REGION Network 32: Sim Bồn 3: Giới hạn mức nước tối thiểu
   RUNG wire#powerrail
      Contact( "AI_HMI_Sim_Mode" )
      { S7_Templates := "SrcType := Real" } LT_Contact(in1 := "AI_LT3213_Bon3_HMI", in2 := 0.0)
      { S7_GenerateENO := "TRUE" } Move(in := 0.0, out1 => "AI_LT3213_Bon3_HMI")
   END_RUNG
   // the same network as SCL:
   IF "AI_HMI_Sim_Mode" AND ("AI_LT3213_Bon3_HMI" < 0.0) THEN "AI_LT3213_Bon3_HMI" := 0.0; END_IF;
END_REGION

REGION Network 33: Sim Bồn 4: Tăng FQ và LT khi dosing
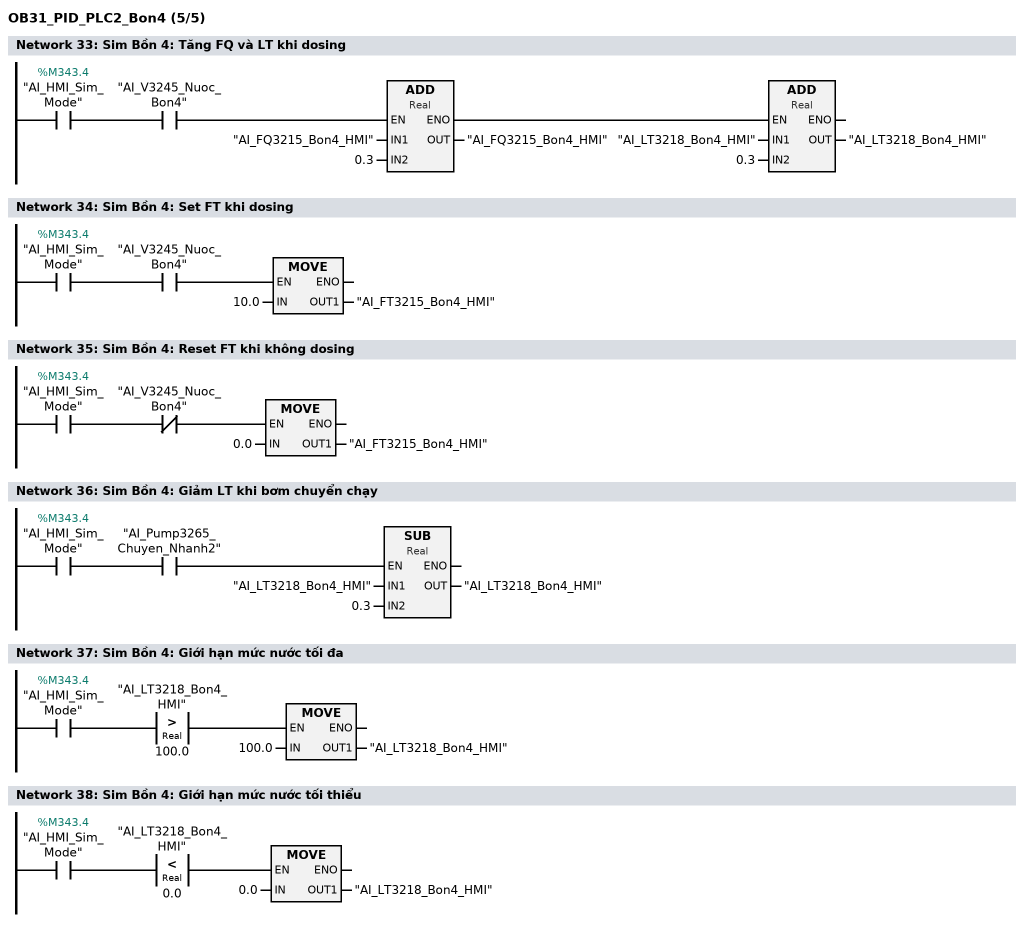
   RUNG wire#powerrail
      Contact( "AI_HMI_Sim_Mode" )
      Contact( "AI_V3245_Nuoc_Bon4" )
      { S7_Templates := "SrcType := Real"; S7_GenerateENO := "TRUE" } Add(in1 := "AI_FQ3215_Bon4_HMI", in2 := 0.3, out => "AI_FQ3215_Bon4_HMI")
      { S7_Templates := "SrcType := Real"; S7_GenerateENO := "TRUE" } Add(in1 := "AI_LT3218_Bon4_HMI", in2 := 0.3, out => "AI_LT3218_Bon4_HMI")
   END_RUNG
   // the same network as SCL:
   // ENO of a box is taken as its EN; it also drops when the box reports an error
   IF "AI_HMI_Sim_Mode" AND "AI_V3245_Nuoc_Bon4" THEN
       "AI_FQ3215_Bon4_HMI" := "AI_FQ3215_Bon4_HMI" + 0.3;
       "AI_LT3218_Bon4_HMI" := "AI_LT3218_Bon4_HMI" + 0.3;
   END_IF;
END_REGION

REGION Network 34: Sim Bồn 4: Set FT khi dosing
   RUNG wire#powerrail
      Contact( "AI_HMI_Sim_Mode" )
      Contact( "AI_V3245_Nuoc_Bon4" )
      { S7_GenerateENO := "TRUE" } Move(in := 10.0, out1 => "AI_FT3215_Bon4_HMI")
   END_RUNG
   // the same network as SCL:
   IF "AI_HMI_Sim_Mode" AND "AI_V3245_Nuoc_Bon4" THEN "AI_FT3215_Bon4_HMI" := 10.0; END_IF;
END_REGION

REGION Network 35: Sim Bồn 4: Reset FT khi không dosing
   RUNG wire#powerrail
      Contact( "AI_HMI_Sim_Mode" )
      I_Contact( "AI_V3245_Nuoc_Bon4" )
      { S7_GenerateENO := "TRUE" } Move(in := 0.0, out1 => "AI_FT3215_Bon4_HMI")
   END_RUNG
   // the same network as SCL:
   IF "AI_HMI_Sim_Mode" AND NOT "AI_V3245_Nuoc_Bon4" THEN "AI_FT3215_Bon4_HMI" := 0.0; END_IF;
END_REGION

REGION Network 36: Sim Bồn 4: Giảm LT khi bơm chuyển chạy
   RUNG wire#powerrail
      Contact( "AI_HMI_Sim_Mode" )
      Contact( "AI_Pump3265_Chuyen_Nhanh2" )
      { S7_Templates := "SrcType := Real"; S7_GenerateENO := "TRUE" } Sub(in1 := "AI_LT3218_Bon4_HMI", in2 := 0.3, out => "AI_LT3218_Bon4_HMI")
   END_RUNG
   // the same network as SCL:
   IF "AI_HMI_Sim_Mode" AND "AI_Pump3265_Chuyen_Nhanh2" THEN
       "AI_LT3218_Bon4_HMI" := "AI_LT3218_Bon4_HMI" - 0.3;
   END_IF;
END_REGION

REGION Network 37: Sim Bồn 4: Giới hạn mức nước tối đa
   RUNG wire#powerrail
      Contact( "AI_HMI_Sim_Mode" )
      { S7_Templates := "SrcType := Real" } GT_Contact(in1 := "AI_LT3218_Bon4_HMI", in2 := 100.0)
      { S7_GenerateENO := "TRUE" } Move(in := 100.0, out1 => "AI_LT3218_Bon4_HMI")
   END_RUNG
   // the same network as SCL:
   IF "AI_HMI_Sim_Mode" AND ("AI_LT3218_Bon4_HMI" > 100.0) THEN "AI_LT3218_Bon4_HMI" := 100.0; END_IF;
END_REGION

REGION Network 38: Sim Bồn 4: Giới hạn mức nước tối thiểu
   RUNG wire#powerrail
      Contact( "AI_HMI_Sim_Mode" )
      { S7_Templates := "SrcType := Real" } LT_Contact(in1 := "AI_LT3218_Bon4_HMI", in2 := 0.0)
      { S7_GenerateENO := "TRUE" } Move(in := 0.0, out1 => "AI_LT3218_Bon4_HMI")
   END_RUNG
   // the same network as SCL:
   IF "AI_HMI_Sim_Mode" AND ("AI_LT3218_Bon4_HMI" < 0.0) THEN "AI_LT3218_Bon4_HMI" := 0.0; END_IF;
END_REGION
END_ORGANIZATION_BLOCK

ORGANIZATION_BLOCK "Cyclic interrupt"   // OB30, LAD, CyclicInterrupt
{ S7_Optimized_Access := 'TRUE' }
VERSION : 0.1
// stored: AutoNumber true, IsIECCheckEnabled false, SetENOAutomatically false
   VAR_INPUT
      Initial_Call : Bool;   // Initial call of this OB
      Event_Count : Int;   // Events discarded
   END_VAR
BEGIN

REGION Network 1
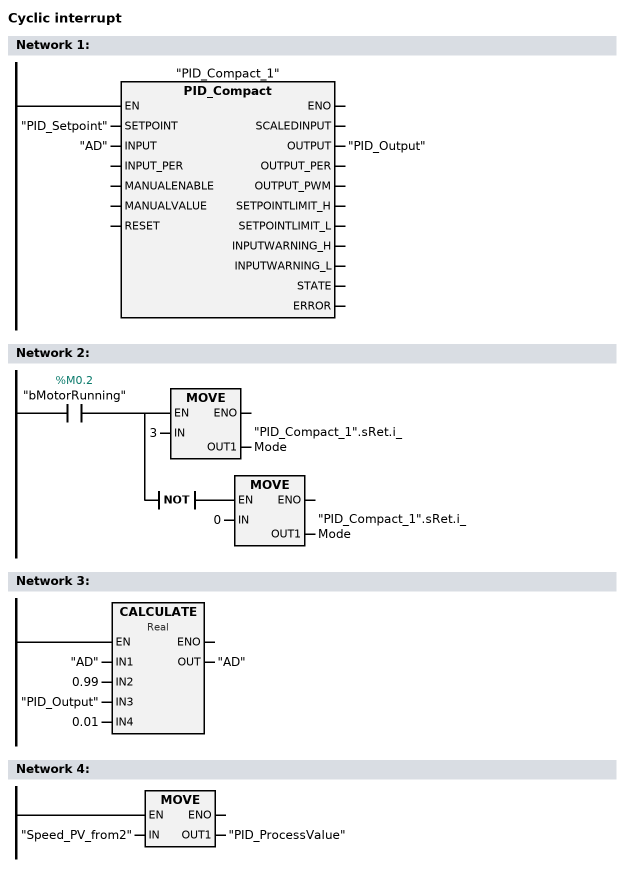
   RUNG wire#powerrail
      "PID_Compact_1".PID_Compact(Setpoint := "PID_Setpoint", Input := "AD", Input_PER :=, ManualEnable :=, ManualValue :=, Reset :=, ScaledInput =>, Output => "PID_Output", Output_PER =>, Output_PWM =>, SetpointLimit_H =>, SetpointLimit_L =>, InputWarning_H =>, InputWarning_L =>, State =>, Error =>)
   END_RUNG
   // the same network as SCL:
   "PID_Compact_1"(Setpoint := "PID_Setpoint", Input := "AD", Output => "PID_Output");   // PID_Compact
END_REGION

REGION Network 2
   RUNG wire#powerrail
      Contact( "bMotorRunning" )
      wire#w1
      Move(in := 3, out1 => "PID_Compact_1".sRet.i_Mode)
   END_RUNG
   RUNG wire#w1
      Not()
      Move(in := 0, out1 => "PID_Compact_1".sRet.i_Mode)
   END_RUNG
   // the same network as SCL:
   IF "bMotorRunning" THEN "PID_Compact_1".sRet.i_Mode := 3; END_IF;
   IF NOT "bMotorRunning" THEN "PID_Compact_1".sRet.i_Mode := 0; END_IF;
END_REGION

REGION Network 3
   RUNG wire#powerrail
      { S7_Templates := "SrcType := Real"; S7_Expression := "IN2*IN1 + IN4*IN3" } Calculate(in1 := "AD", in2 := 0.99, in3 := "PID_Output", in4 := 0.01, out => "AD")
   END_RUNG
   // the same network as SCL:
   "AD" := 0.99*"AD" + 0.01*"PID_Output";
END_REGION

REGION Network 4
   RUNG wire#powerrail
      Move(in := "Speed_PV_from2", out1 => "PID_ProcessValue")
   END_RUNG
   // the same network as SCL:
   "PID_ProcessValue" := "Speed_PV_from2";
END_REGION
END_ORGANIZATION_BLOCK

ORGANIZATION_BLOCK "OB30_Encoder_100ms"   // OB30, LAD, CyclicInterrupt
{ S7_Optimized_Access := 'TRUE' }
VERSION : 0.1
// stored: AutoNumber true, IsIECCheckEnabled false, SetENOAutomatically false
   VAR_INPUT
      Initial_Call : Bool;   // Initial call of this OB
      Event_Count : Int;   // Events discarded
   END_VAR
BEGIN

REGION Network 1: Đọc giá trị HSC và tính Delta Count
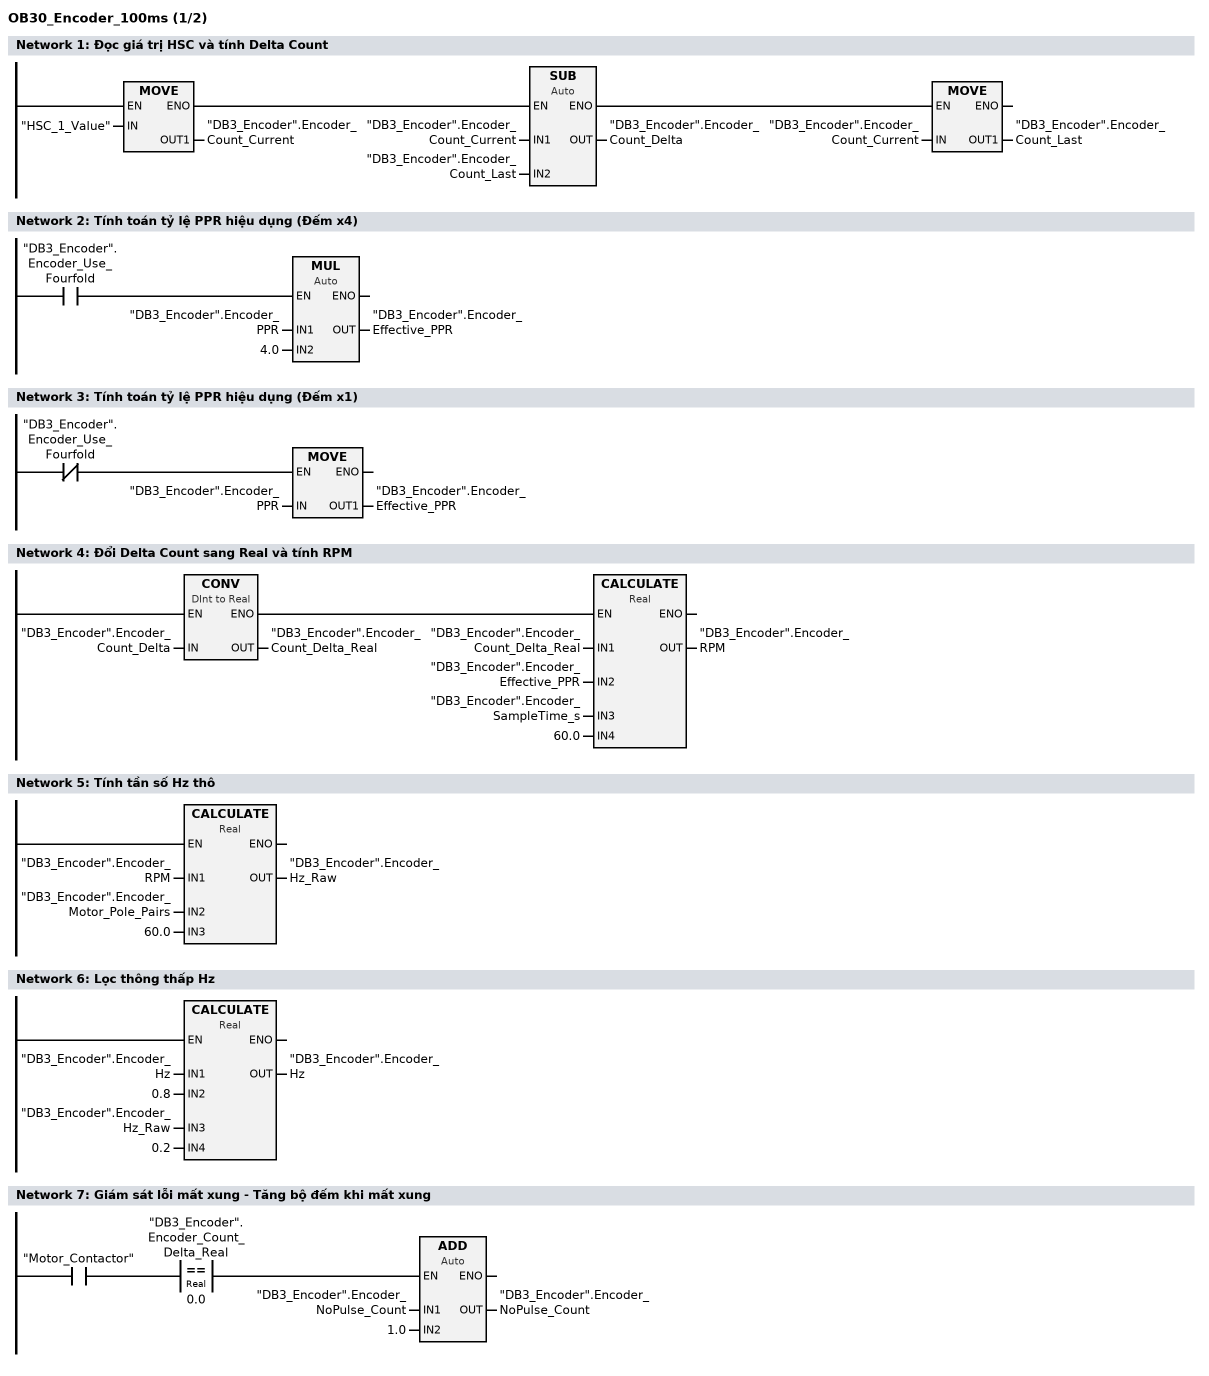
   RUNG wire#powerrail
      { S7_GenerateENO := "TRUE" } Move(in := "HSC_1_Value", out1 => "DB3_Encoder".Encoder_Count_Current)
      { S7_GenerateENO := "TRUE" } Sub(in1 := "DB3_Encoder".Encoder_Count_Current, in2 := "DB3_Encoder".Encoder_Count_Last, out => "DB3_Encoder".Encoder_Count_Delta)
      { S7_GenerateENO := "TRUE" } Move(in := "DB3_Encoder".Encoder_Count_Current, out1 => "DB3_Encoder".Encoder_Count_Last)
   END_RUNG
   // the same network as SCL:
   // ENO of a box is taken as its EN; it also drops when the box reports an error
   "DB3_Encoder".Encoder_Count_Current := "HSC_1_Value";
   "DB3_Encoder".Encoder_Count_Delta := "DB3_Encoder".Encoder_Count_Current - "DB3_Encoder".Encoder_Count_Last;
   "DB3_Encoder".Encoder_Count_Last := "DB3_Encoder".Encoder_Count_Current;
END_REGION

REGION Network 2: Tính toán tỷ lệ PPR hiệu dụng (Đếm x4)
   RUNG wire#powerrail
      Contact( "DB3_Encoder".Encoder_Use_Fourfold )
      { S7_GenerateENO := "TRUE" } Mul(in1 := "DB3_Encoder".Encoder_PPR, in2 := 4.0, out => "DB3_Encoder".Encoder_Effective_PPR)
   END_RUNG
   // the same network as SCL:
   IF "DB3_Encoder".Encoder_Use_Fourfold THEN
       "DB3_Encoder".Encoder_Effective_PPR := "DB3_Encoder".Encoder_PPR * 4.0;
   END_IF;
END_REGION

REGION Network 3: Tính toán tỷ lệ PPR hiệu dụng (Đếm x1)
   RUNG wire#powerrail
      I_Contact( "DB3_Encoder".Encoder_Use_Fourfold )
      { S7_GenerateENO := "TRUE" } Move(in := "DB3_Encoder".Encoder_PPR, out1 => "DB3_Encoder".Encoder_Effective_PPR)
   END_RUNG
   // the same network as SCL:
   IF NOT "DB3_Encoder".Encoder_Use_Fourfold THEN
       "DB3_Encoder".Encoder_Effective_PPR := "DB3_Encoder".Encoder_PPR;
   END_IF;
END_REGION

REGION Network 4: Đổi Delta Count sang Real và tính RPM
   RUNG wire#powerrail
      { S7_Templates := "[SrcType := DInt, DestType := Real]"; S7_GenerateENO := "TRUE" } Convert(in := "DB3_Encoder".Encoder_Count_Delta, out => "DB3_Encoder".Encoder_Count_Delta_Real)
      { S7_Templates := "SrcType := Real"; S7_GenerateENO := "TRUE"; S7_Expression := "(IN1 * IN4) / (IN2 * IN3)" } Calculate(in1 := "DB3_Encoder".Encoder_Count_Delta_Real, in2 := "DB3_Encoder".Encoder_Effective_PPR, in3 := "DB3_Encoder".Encoder_SampleTime_s, in4 := 60.0, out => "DB3_Encoder".Encoder_RPM)
   END_RUNG
   // the same network as SCL:
   // ENO of a box is taken as its EN; it also drops when the box reports an error
   "DB3_Encoder".Encoder_Count_Delta_Real := DINT_TO_REAL("DB3_Encoder".Encoder_Count_Delta);
   "DB3_Encoder".Encoder_RPM := ("DB3_Encoder".Encoder_Count_Delta_Real * 60.0) / ("DB3_Encoder".Encoder_Effective_PPR * "DB3_Encoder".Encoder_SampleTime_s);
END_REGION

REGION Network 5: Tính tần số Hz thô
   RUNG wire#powerrail
      { S7_Templates := "SrcType := Real"; S7_GenerateENO := "TRUE"; S7_Expression := "(IN1 * IN2) / IN3" } Calculate(in1 := "DB3_Encoder".Encoder_RPM, in2 := "DB3_Encoder".Encoder_Motor_Pole_Pairs, in3 := 60.0, out => "DB3_Encoder".Encoder_Hz_Raw)
   END_RUNG
   // the same network as SCL:
   "DB3_Encoder".Encoder_Hz_Raw := ("DB3_Encoder".Encoder_RPM * "DB3_Encoder".Encoder_Motor_Pole_Pairs) / 60.0;
END_REGION

REGION Network 6: Lọc thông thấp Hz
   RUNG wire#powerrail
      { S7_Templates := "SrcType := Real"; S7_GenerateENO := "TRUE"; S7_Expression := "(IN1 * IN2) + (IN3 * IN4)" } Calculate(in1 := "DB3_Encoder".Encoder_Hz, in2 := 0.8, in3 := "DB3_Encoder".Encoder_Hz_Raw, in4 := 0.2, out => "DB3_Encoder".Encoder_Hz)
   END_RUNG
   // the same network as SCL:
   "DB3_Encoder".Encoder_Hz := ("DB3_Encoder".Encoder_Hz * 0.8) + ("DB3_Encoder".Encoder_Hz_Raw * 0.2);
END_REGION

REGION Network 7: Giám sát lỗi mất xung - Tăng bộ đếm khi mất xung
   RUNG wire#powerrail
      Contact( "Motor_Contactor" )
      { S7_Templates := "SrcType := Real" } EQ_Contact(in1 := "DB3_Encoder".Encoder_Count_Delta_Real, in2 := 0.0)
      { S7_GenerateENO := "TRUE" } Add(in1 := "DB3_Encoder".Encoder_NoPulse_Count, in2 := 1.0, out => "DB3_Encoder".Encoder_NoPulse_Count)
   END_RUNG
   // the same network as SCL:
   IF "Motor_Contactor" AND ("DB3_Encoder".Encoder_Count_Delta_Real = 0.0) THEN
       "DB3_Encoder".Encoder_NoPulse_Count := "DB3_Encoder".Encoder_NoPulse_Count + 1.0;
   END_IF;
END_REGION

REGION Network 8: Giám sát lỗi mất xung - Reset bộ đếm khi có xung
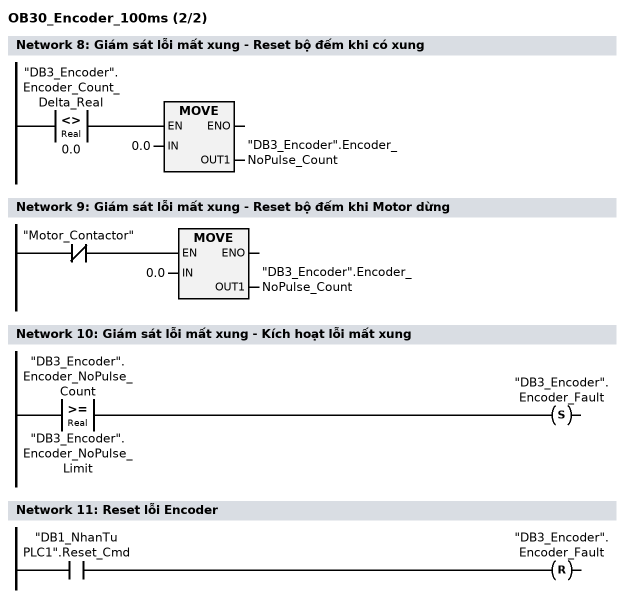
   RUNG wire#powerrail
      { S7_Templates := "SrcType := Real" } NE_Contact(in1 := "DB3_Encoder".Encoder_Count_Delta_Real, in2 := 0.0)
      { S7_GenerateENO := "TRUE" } Move(in := 0.0, out1 => "DB3_Encoder".Encoder_NoPulse_Count)
   END_RUNG
   // the same network as SCL:
   IF "DB3_Encoder".Encoder_Count_Delta_Real <> 0.0 THEN "DB3_Encoder".Encoder_NoPulse_Count := 0.0; END_IF;
END_REGION

REGION Network 9: Giám sát lỗi mất xung - Reset bộ đếm khi Motor dừng
   RUNG wire#powerrail
      I_Contact( "Motor_Contactor" )
      { S7_GenerateENO := "TRUE" } Move(in := 0.0, out1 => "DB3_Encoder".Encoder_NoPulse_Count)
   END_RUNG
   // the same network as SCL:
   IF NOT "Motor_Contactor" THEN "DB3_Encoder".Encoder_NoPulse_Count := 0.0; END_IF;
END_REGION

REGION Network 10: Giám sát lỗi mất xung - Kích hoạt lỗi mất xung
   RUNG wire#powerrail
      { S7_Templates := "SrcType := Real" } GE_Contact(in1 := "DB3_Encoder".Encoder_NoPulse_Count, in2 := "DB3_Encoder".Encoder_NoPulse_Limit)
      S_Coil( "DB3_Encoder".Encoder_Fault )
   END_RUNG
   // the same network as SCL:
   IF "DB3_Encoder".Encoder_NoPulse_Count >= "DB3_Encoder".Encoder_NoPulse_Limit THEN
       "DB3_Encoder".Encoder_Fault := TRUE;
   END_IF;
END_REGION

REGION Network 11: Reset lỗi Encoder
   RUNG wire#powerrail
      Contact( "DB1_NhanTuPLC1".Reset_Cmd )
      R_Coil( "DB3_Encoder".Encoder_Fault )
   END_RUNG
   // the same network as SCL:
   IF "DB1_NhanTuPLC1".Reset_Cmd THEN "DB3_Encoder".Encoder_Fault := FALSE; END_IF;
END_REGION
END_ORGANIZATION_BLOCK

FUNCTION "FC_SCADA_Simulation" : Void   // FC10, LAD
{ S7_Optimized_Access := 'TRUE' }
VERSION : 0.1
// stored: AutoNumber true, IsIECCheckEnabled false
BEGIN

REGION Network 1: Tạo xung kích hoạt chu kỳ mô phỏng (50ms)
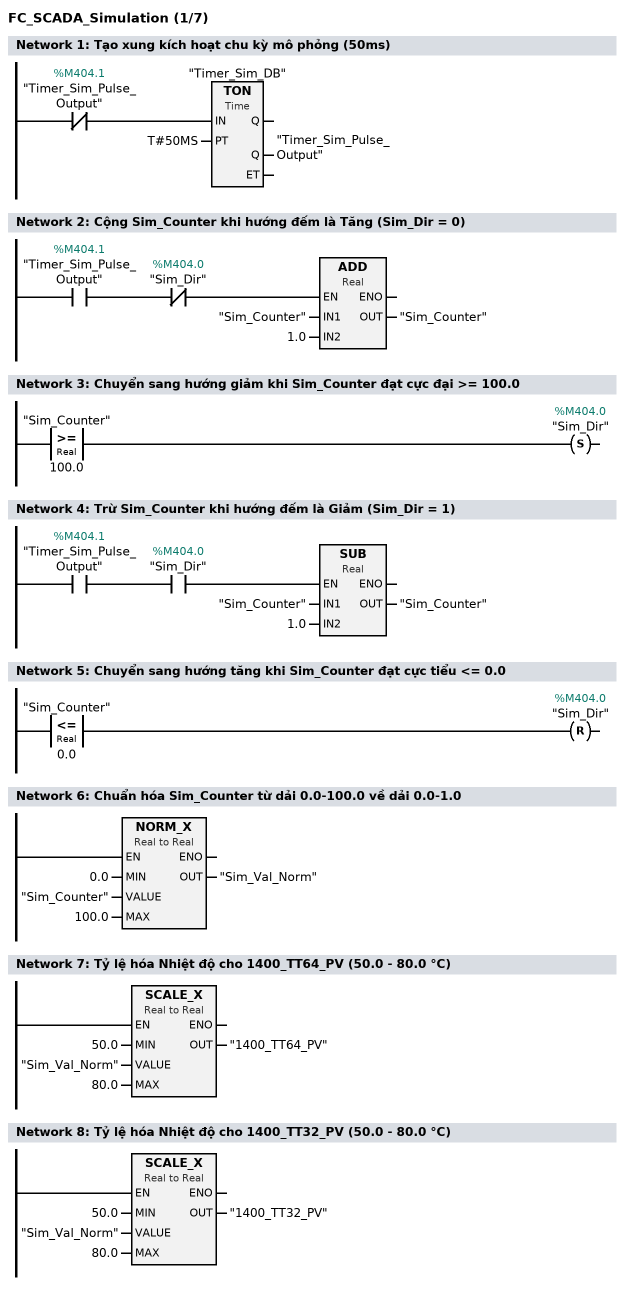
   RUNG wire#powerrail
      I_Contact( "Timer_Sim_Pulse_Output" )
      { S7_Templates := "time_type := Time" } "Timer_Sim_DB".TON(pt := T#50MS, q => "Timer_Sim_Pulse_Output", et =>)
   END_RUNG
   // the same network as SCL:
   "Timer_Sim_DB".TON(IN := NOT "Timer_Sim_Pulse_Output", PT := T#50MS, Q => "Timer_Sim_Pulse_Output");
END_REGION

REGION Network 2: Cộng Sim_Counter khi hướng đếm là Tăng (Sim_Dir = 0)
   RUNG wire#powerrail
      Contact( "Timer_Sim_Pulse_Output" )
      I_Contact( "Sim_Dir" )
      { S7_Templates := "SrcType := Real"; S7_GenerateENO := "TRUE" } Add(in1 := "Sim_Counter", in2 := 1.0, out => "Sim_Counter")
   END_RUNG
   // the same network as SCL:
   IF "Timer_Sim_Pulse_Output" AND NOT "Sim_Dir" THEN "Sim_Counter" := "Sim_Counter" + 1.0; END_IF;
END_REGION

REGION Network 3: Chuyển sang hướng giảm khi Sim_Counter đạt cực đại >= 100.0
   RUNG wire#powerrail
      { S7_Templates := "SrcType := Real" } GE_Contact(in1 := "Sim_Counter", in2 := 100.0)
      S_Coil( "Sim_Dir" )
   END_RUNG
   // the same network as SCL:
   IF "Sim_Counter" >= 100.0 THEN "Sim_Dir" := TRUE; END_IF;
END_REGION

REGION Network 4: Trừ Sim_Counter khi hướng đếm là Giảm (Sim_Dir = 1)
   RUNG wire#powerrail
      Contact( "Timer_Sim_Pulse_Output" )
      Contact( "Sim_Dir" )
      { S7_Templates := "SrcType := Real"; S7_GenerateENO := "TRUE" } Sub(in1 := "Sim_Counter", in2 := 1.0, out => "Sim_Counter")
   END_RUNG
   // the same network as SCL:
   IF "Timer_Sim_Pulse_Output" AND "Sim_Dir" THEN "Sim_Counter" := "Sim_Counter" - 1.0; END_IF;
END_REGION

REGION Network 5: Chuyển sang hướng tăng khi Sim_Counter đạt cực tiểu <= 0.0
   RUNG wire#powerrail
      { S7_Templates := "SrcType := Real" } LE_Contact(in1 := "Sim_Counter", in2 := 0.0)
      R_Coil( "Sim_Dir" )
   END_RUNG
   // the same network as SCL:
   IF "Sim_Counter" <= 0.0 THEN "Sim_Dir" := FALSE; END_IF;
END_REGION

REGION Network 6: Chuẩn hóa Sim_Counter từ dải 0.0-100.0 về dải 0.0-1.0
   RUNG wire#powerrail
      { S7_Templates := "[SrcType := Real, DestType := Real]" } Normalize(min := 0.0, value := "Sim_Counter", max := 100.0, out => "Sim_Val_Norm")
   END_RUNG
   // the same network as SCL:
   "Sim_Val_Norm" := NORM_X(MIN := 0.0, VALUE := "Sim_Counter", MAX := 100.0);
END_REGION

REGION Network 7: Tỷ lệ hóa Nhiệt độ cho 1400_TT64_PV (50.0 - 80.0 °C)
   RUNG wire#powerrail
      { S7_Templates := "[SrcType := Real, DestType := Real]" } Scale(min := 50.0, value := "Sim_Val_Norm", max := 80.0, out => "1400_TT64_PV")
   END_RUNG
   // the same network as SCL:
   "1400_TT64_PV" := SCALE_X(MIN := 50.0, VALUE := "Sim_Val_Norm", MAX := 80.0);
END_REGION

REGION Network 8: Tỷ lệ hóa Nhiệt độ cho 1400_TT32_PV (50.0 - 80.0 °C)
   RUNG wire#powerrail
      { S7_Templates := "[SrcType := Real, DestType := Real]" } Scale(min := 50.0, value := "Sim_Val_Norm", max := 80.0, out => "1400_TT32_PV")
   END_RUNG
   // the same network as SCL:
   "1400_TT32_PV" := SCALE_X(MIN := 50.0, VALUE := "Sim_Val_Norm", MAX := 80.0);
END_REGION

REGION Network 9: Tỷ lệ hóa Nhiệt độ cho 1400_TT101_PV (50.0 - 80.0 °C)
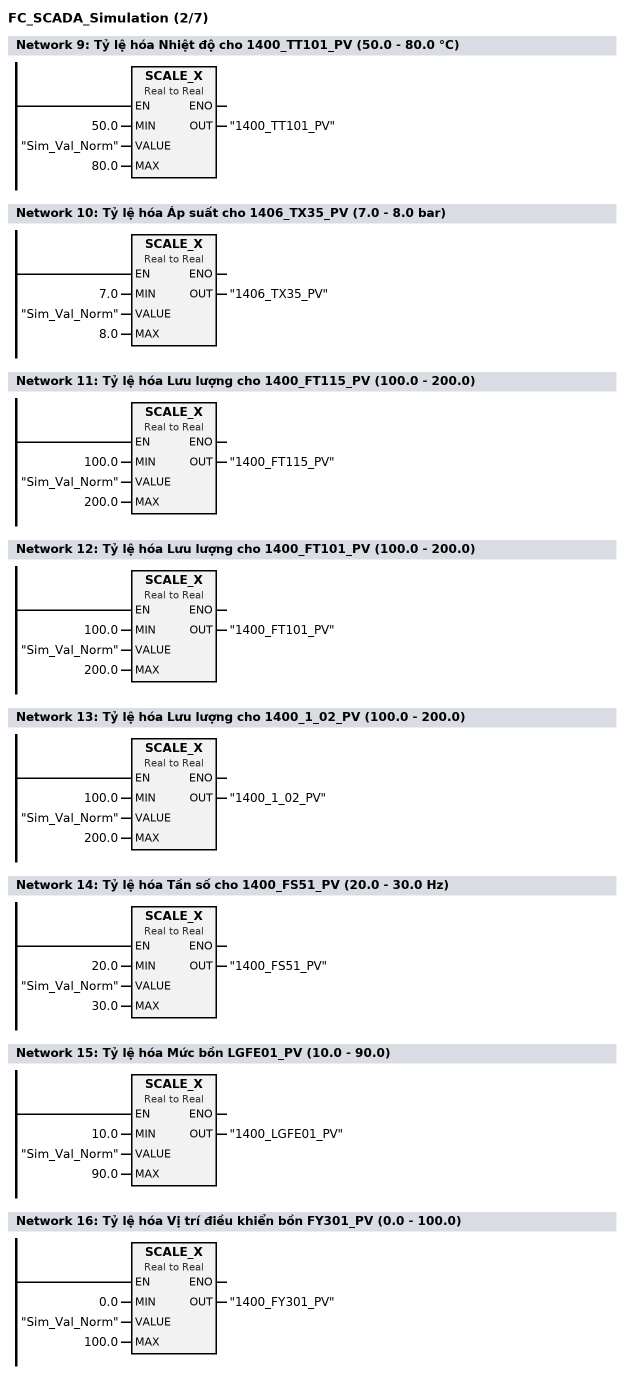
   RUNG wire#powerrail
      { S7_Templates := "[SrcType := Real, DestType := Real]" } Scale(min := 50.0, value := "Sim_Val_Norm", max := 80.0, out => "1400_TT101_PV")
   END_RUNG
   // the same network as SCL:
   "1400_TT101_PV" := SCALE_X(MIN := 50.0, VALUE := "Sim_Val_Norm", MAX := 80.0);
END_REGION

REGION Network 10: Tỷ lệ hóa Áp suất cho 1406_TX35_PV (7.0 - 8.0 bar)
   RUNG wire#powerrail
      { S7_Templates := "[SrcType := Real, DestType := Real]" } Scale(min := 7.0, value := "Sim_Val_Norm", max := 8.0, out => "1406_TX35_PV")
   END_RUNG
   // the same network as SCL:
   "1406_TX35_PV" := SCALE_X(MIN := 7.0, VALUE := "Sim_Val_Norm", MAX := 8.0);
END_REGION

REGION Network 11: Tỷ lệ hóa Lưu lượng cho 1400_FT115_PV (100.0 - 200.0)
   RUNG wire#powerrail
      { S7_Templates := "[SrcType := Real, DestType := Real]" } Scale(min := 100.0, value := "Sim_Val_Norm", max := 200.0, out => "1400_FT115_PV")
   END_RUNG
   // the same network as SCL:
   "1400_FT115_PV" := SCALE_X(MIN := 100.0, VALUE := "Sim_Val_Norm", MAX := 200.0);
END_REGION

REGION Network 12: Tỷ lệ hóa Lưu lượng cho 1400_FT101_PV (100.0 - 200.0)
   RUNG wire#powerrail
      { S7_Templates := "[SrcType := Real, DestType := Real]" } Scale(min := 100.0, value := "Sim_Val_Norm", max := 200.0, out => "1400_FT101_PV")
   END_RUNG
   // the same network as SCL:
   "1400_FT101_PV" := SCALE_X(MIN := 100.0, VALUE := "Sim_Val_Norm", MAX := 200.0);
END_REGION

REGION Network 13: Tỷ lệ hóa Lưu lượng cho 1400_1_02_PV (100.0 - 200.0)
   RUNG wire#powerrail
      { S7_Templates := "[SrcType := Real, DestType := Real]" } Scale(min := 100.0, value := "Sim_Val_Norm", max := 200.0, out => "1400_1_02_PV")
   END_RUNG
   // the same network as SCL:
   "1400_1_02_PV" := SCALE_X(MIN := 100.0, VALUE := "Sim_Val_Norm", MAX := 200.0);
END_REGION

REGION Network 14: Tỷ lệ hóa Tần số cho 1400_FS51_PV (20.0 - 30.0 Hz)
   RUNG wire#powerrail
      { S7_Templates := "[SrcType := Real, DestType := Real]" } Scale(min := 20.0, value := "Sim_Val_Norm", max := 30.0, out => "1400_FS51_PV")
   END_RUNG
   // the same network as SCL:
   "1400_FS51_PV" := SCALE_X(MIN := 20.0, VALUE := "Sim_Val_Norm", MAX := 30.0);
END_REGION

REGION Network 15: Tỷ lệ hóa Mức bồn LGFE01_PV (10.0 - 90.0)
   RUNG wire#powerrail
      { S7_Templates := "[SrcType := Real, DestType := Real]" } Scale(min := 10.0, value := "Sim_Val_Norm", max := 90.0, out => "1400_LGFE01_PV")
   END_RUNG
   // the same network as SCL:
   "1400_LGFE01_PV" := SCALE_X(MIN := 10.0, VALUE := "Sim_Val_Norm", MAX := 90.0);
END_REGION

REGION Network 16: Tỷ lệ hóa Vị trí điều khiển bồn FY301_PV (0.0 - 100.0)
   RUNG wire#powerrail
      { S7_Templates := "[SrcType := Real, DestType := Real]" } Scale(min := 0.0, value := "Sim_Val_Norm", max := 100.0, out => "1400_FY301_PV")
   END_RUNG
   // the same network as SCL:
   "1400_FY301_PV" := SCALE_X(MIN := 0.0, VALUE := "Sim_Val_Norm", MAX := 100.0);
END_REGION

REGION Network 17: Tỷ lệ hóa FTT02_PV (40.0 - 70.0)
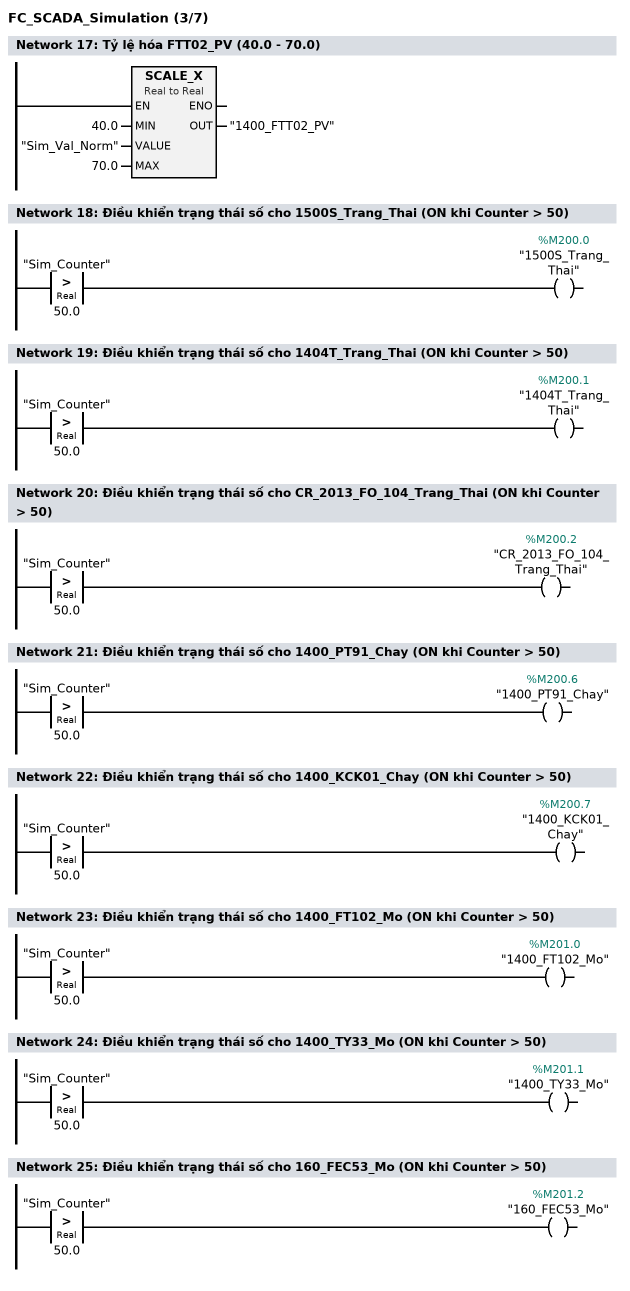
   RUNG wire#powerrail
      { S7_Templates := "[SrcType := Real, DestType := Real]" } Scale(min := 40.0, value := "Sim_Val_Norm", max := 70.0, out => "1400_FTT02_PV")
   END_RUNG
   // the same network as SCL:
   "1400_FTT02_PV" := SCALE_X(MIN := 40.0, VALUE := "Sim_Val_Norm", MAX := 70.0);
END_REGION

REGION Network 18: Điều khiển trạng thái số cho 1500S_Trang_Thai (ON khi Counter > 50)
   RUNG wire#powerrail
      { S7_Templates := "SrcType := Real" } GT_Contact(in1 := "Sim_Counter", in2 := 50.0)
      Coil( "1500S_Trang_Thai" )
   END_RUNG
   // the same network as SCL:
   "1500S_Trang_Thai" := "Sim_Counter" > 50.0;
END_REGION

REGION Network 19: Điều khiển trạng thái số cho 1404T_Trang_Thai (ON khi Counter > 50)
   RUNG wire#powerrail
      { S7_Templates := "SrcType := Real" } GT_Contact(in1 := "Sim_Counter", in2 := 50.0)
      Coil( "1404T_Trang_Thai" )
   END_RUNG
   // the same network as SCL:
   "1404T_Trang_Thai" := "Sim_Counter" > 50.0;
END_REGION

REGION Network 20: Điều khiển trạng thái số cho CR_2013_FO_104_Trang_Thai (ON khi Counter > 50)
   RUNG wire#powerrail
      { S7_Templates := "SrcType := Real" } GT_Contact(in1 := "Sim_Counter", in2 := 50.0)
      Coil( "CR_2013_FO_104_Trang_Thai" )
   END_RUNG
   // the same network as SCL:
   "CR_2013_FO_104_Trang_Thai" := "Sim_Counter" > 50.0;
END_REGION

REGION Network 21: Điều khiển trạng thái số cho 1400_PT91_Chay (ON khi Counter > 50)
   RUNG wire#powerrail
      { S7_Templates := "SrcType := Real" } GT_Contact(in1 := "Sim_Counter", in2 := 50.0)
      Coil( "1400_PT91_Chay" )
   END_RUNG
   // the same network as SCL:
   "1400_PT91_Chay" := "Sim_Counter" > 50.0;
END_REGION

REGION Network 22: Điều khiển trạng thái số cho 1400_KCK01_Chay (ON khi Counter > 50)
   RUNG wire#powerrail
      { S7_Templates := "SrcType := Real" } GT_Contact(in1 := "Sim_Counter", in2 := 50.0)
      Coil( "1400_KCK01_Chay" )
   END_RUNG
   // the same network as SCL:
   "1400_KCK01_Chay" := "Sim_Counter" > 50.0;
END_REGION

REGION Network 23: Điều khiển trạng thái số cho 1400_FT102_Mo (ON khi Counter > 50)
   RUNG wire#powerrail
      { S7_Templates := "SrcType := Real" } GT_Contact(in1 := "Sim_Counter", in2 := 50.0)
      Coil( "1400_FT102_Mo" )
   END_RUNG
   // the same network as SCL:
   "1400_FT102_Mo" := "Sim_Counter" > 50.0;
END_REGION

REGION Network 24: Điều khiển trạng thái số cho 1400_TY33_Mo (ON khi Counter > 50)
   RUNG wire#powerrail
      { S7_Templates := "SrcType := Real" } GT_Contact(in1 := "Sim_Counter", in2 := 50.0)
      Coil( "1400_TY33_Mo" )
   END_RUNG
   // the same network as SCL:
   "1400_TY33_Mo" := "Sim_Counter" > 50.0;
END_REGION

REGION Network 25: Điều khiển trạng thái số cho 160_FEC53_Mo (ON khi Counter > 50)
   RUNG wire#powerrail
      { S7_Templates := "SrcType := Real" } GT_Contact(in1 := "Sim_Counter", in2 := 50.0)
      Coil( "160_FEC53_Mo" )
   END_RUNG
   // the same network as SCL:
   "160_FEC53_Mo" := "Sim_Counter" > 50.0;
END_REGION

REGION Network 26: Điều khiển trạng thái số cho BFOC_SS_20_06_Trang_Thai (ON khi Counter <= 50)
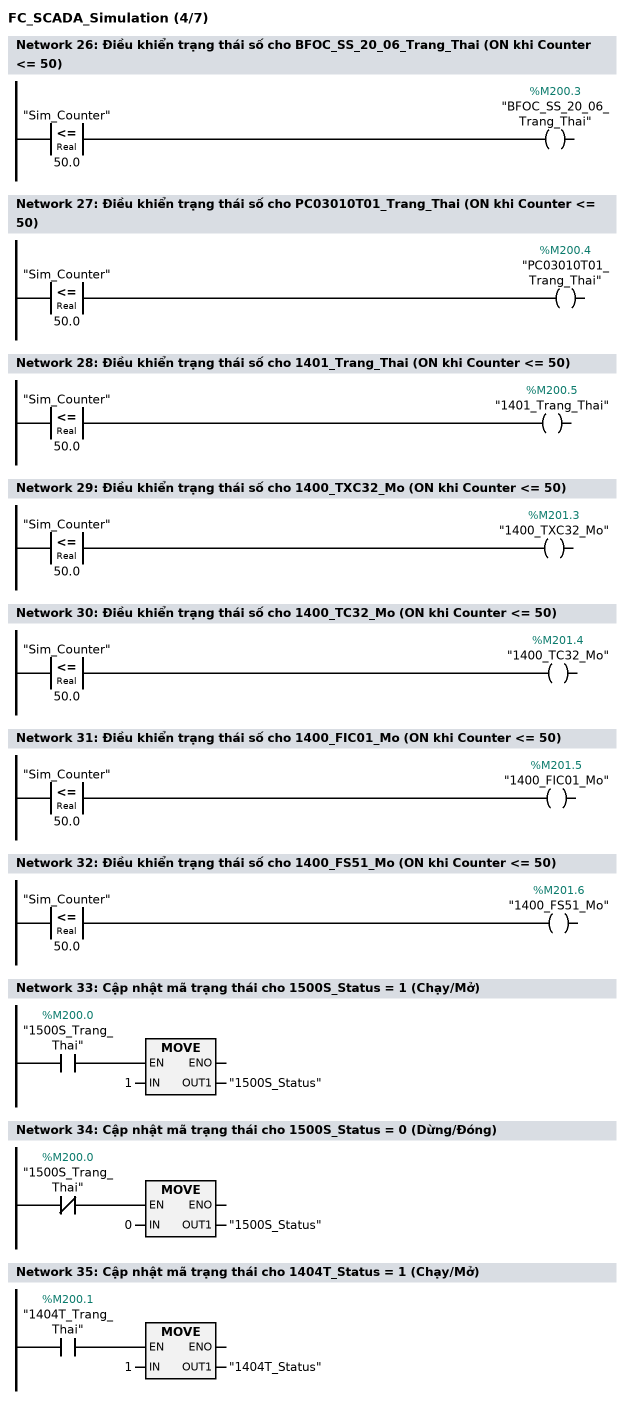
   RUNG wire#powerrail
      { S7_Templates := "SrcType := Real" } LE_Contact(in1 := "Sim_Counter", in2 := 50.0)
      Coil( "BFOC_SS_20_06_Trang_Thai" )
   END_RUNG
   // the same network as SCL:
   "BFOC_SS_20_06_Trang_Thai" := "Sim_Counter" <= 50.0;
END_REGION

REGION Network 27: Điều khiển trạng thái số cho PC03010T01_Trang_Thai (ON khi Counter <= 50)
   RUNG wire#powerrail
      { S7_Templates := "SrcType := Real" } LE_Contact(in1 := "Sim_Counter", in2 := 50.0)
      Coil( "PC03010T01_Trang_Thai" )
   END_RUNG
   // the same network as SCL:
   "PC03010T01_Trang_Thai" := "Sim_Counter" <= 50.0;
END_REGION

REGION Network 28: Điều khiển trạng thái số cho 1401_Trang_Thai (ON khi Counter <= 50)
   RUNG wire#powerrail
      { S7_Templates := "SrcType := Real" } LE_Contact(in1 := "Sim_Counter", in2 := 50.0)
      Coil( "1401_Trang_Thai" )
   END_RUNG
   // the same network as SCL:
   "1401_Trang_Thai" := "Sim_Counter" <= 50.0;
END_REGION

REGION Network 29: Điều khiển trạng thái số cho 1400_TXC32_Mo (ON khi Counter <= 50)
   RUNG wire#powerrail
      { S7_Templates := "SrcType := Real" } LE_Contact(in1 := "Sim_Counter", in2 := 50.0)
      Coil( "1400_TXC32_Mo" )
   END_RUNG
   // the same network as SCL:
   "1400_TXC32_Mo" := "Sim_Counter" <= 50.0;
END_REGION

REGION Network 30: Điều khiển trạng thái số cho 1400_TC32_Mo (ON khi Counter <= 50)
   RUNG wire#powerrail
      { S7_Templates := "SrcType := Real" } LE_Contact(in1 := "Sim_Counter", in2 := 50.0)
      Coil( "1400_TC32_Mo" )
   END_RUNG
   // the same network as SCL:
   "1400_TC32_Mo" := "Sim_Counter" <= 50.0;
END_REGION

REGION Network 31: Điều khiển trạng thái số cho 1400_FIC01_Mo (ON khi Counter <= 50)
   RUNG wire#powerrail
      { S7_Templates := "SrcType := Real" } LE_Contact(in1 := "Sim_Counter", in2 := 50.0)
      Coil( "1400_FIC01_Mo" )
   END_RUNG
   // the same network as SCL:
   "1400_FIC01_Mo" := "Sim_Counter" <= 50.0;
END_REGION

REGION Network 32: Điều khiển trạng thái số cho 1400_FS51_Mo (ON khi Counter <= 50)
   RUNG wire#powerrail
      { S7_Templates := "SrcType := Real" } LE_Contact(in1 := "Sim_Counter", in2 := 50.0)
      Coil( "1400_FS51_Mo" )
   END_RUNG
   // the same network as SCL:
   "1400_FS51_Mo" := "Sim_Counter" <= 50.0;
END_REGION

REGION Network 33: Cập nhật mã trạng thái cho 1500S_Status = 1 (Chạy/Mở)
   RUNG wire#powerrail
      Contact( "1500S_Trang_Thai" )
      { S7_GenerateENO := "TRUE" } Move(in := 1, out1 => "1500S_Status")
   END_RUNG
   // the same network as SCL:
   IF "1500S_Trang_Thai" THEN "1500S_Status" := 1; END_IF;
END_REGION

REGION Network 34: Cập nhật mã trạng thái cho 1500S_Status = 0 (Dừng/Đóng)
   RUNG wire#powerrail
      I_Contact( "1500S_Trang_Thai" )
      { S7_GenerateENO := "TRUE" } Move(in := 0, out1 => "1500S_Status")
   END_RUNG
   // the same network as SCL:
   IF NOT "1500S_Trang_Thai" THEN "1500S_Status" := 0; END_IF;
END_REGION

REGION Network 35: Cập nhật mã trạng thái cho 1404T_Status = 1 (Chạy/Mở)
   RUNG wire#powerrail
      Contact( "1404T_Trang_Thai" )
      { S7_GenerateENO := "TRUE" } Move(in := 1, out1 => "1404T_Status")
   END_RUNG
   // the same network as SCL:
   IF "1404T_Trang_Thai" THEN "1404T_Status" := 1; END_IF;
END_REGION

REGION Network 36: Cập nhật mã trạng thái cho 1404T_Status = 0 (Dừng/Đóng)
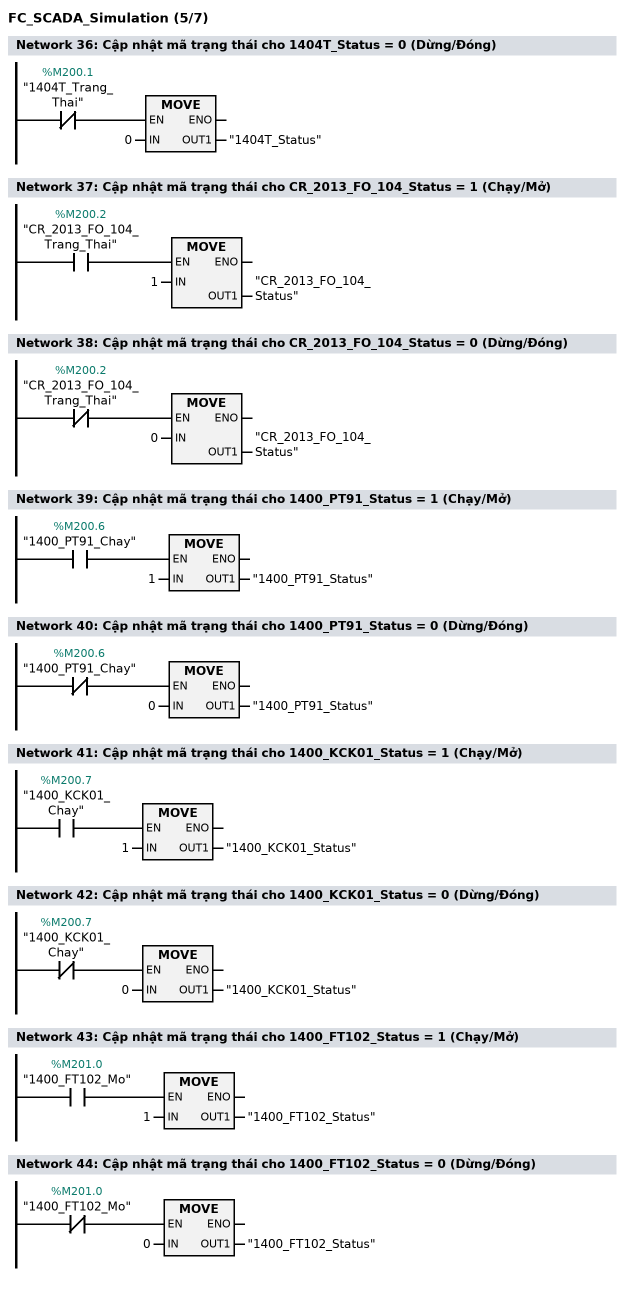
   RUNG wire#powerrail
      I_Contact( "1404T_Trang_Thai" )
      { S7_GenerateENO := "TRUE" } Move(in := 0, out1 => "1404T_Status")
   END_RUNG
   // the same network as SCL:
   IF NOT "1404T_Trang_Thai" THEN "1404T_Status" := 0; END_IF;
END_REGION

REGION Network 37: Cập nhật mã trạng thái cho CR_2013_FO_104_Status = 1 (Chạy/Mở)
   RUNG wire#powerrail
      Contact( "CR_2013_FO_104_Trang_Thai" )
      { S7_GenerateENO := "TRUE" } Move(in := 1, out1 => "CR_2013_FO_104_Status")
   END_RUNG
   // the same network as SCL:
   IF "CR_2013_FO_104_Trang_Thai" THEN "CR_2013_FO_104_Status" := 1; END_IF;
END_REGION

REGION Network 38: Cập nhật mã trạng thái cho CR_2013_FO_104_Status = 0 (Dừng/Đóng)
   RUNG wire#powerrail
      I_Contact( "CR_2013_FO_104_Trang_Thai" )
      { S7_GenerateENO := "TRUE" } Move(in := 0, out1 => "CR_2013_FO_104_Status")
   END_RUNG
   // the same network as SCL:
   IF NOT "CR_2013_FO_104_Trang_Thai" THEN "CR_2013_FO_104_Status" := 0; END_IF;
END_REGION

REGION Network 39: Cập nhật mã trạng thái cho 1400_PT91_Status = 1 (Chạy/Mở)
   RUNG wire#powerrail
      Contact( "1400_PT91_Chay" )
      { S7_GenerateENO := "TRUE" } Move(in := 1, out1 => "1400_PT91_Status")
   END_RUNG
   // the same network as SCL:
   IF "1400_PT91_Chay" THEN "1400_PT91_Status" := 1; END_IF;
END_REGION

REGION Network 40: Cập nhật mã trạng thái cho 1400_PT91_Status = 0 (Dừng/Đóng)
   RUNG wire#powerrail
      I_Contact( "1400_PT91_Chay" )
      { S7_GenerateENO := "TRUE" } Move(in := 0, out1 => "1400_PT91_Status")
   END_RUNG
   // the same network as SCL:
   IF NOT "1400_PT91_Chay" THEN "1400_PT91_Status" := 0; END_IF;
END_REGION

REGION Network 41: Cập nhật mã trạng thái cho 1400_KCK01_Status = 1 (Chạy/Mở)
   RUNG wire#powerrail
      Contact( "1400_KCK01_Chay" )
      { S7_GenerateENO := "TRUE" } Move(in := 1, out1 => "1400_KCK01_Status")
   END_RUNG
   // the same network as SCL:
   IF "1400_KCK01_Chay" THEN "1400_KCK01_Status" := 1; END_IF;
END_REGION

REGION Network 42: Cập nhật mã trạng thái cho 1400_KCK01_Status = 0 (Dừng/Đóng)
   RUNG wire#powerrail
      I_Contact( "1400_KCK01_Chay" )
      { S7_GenerateENO := "TRUE" } Move(in := 0, out1 => "1400_KCK01_Status")
   END_RUNG
   // the same network as SCL:
   IF NOT "1400_KCK01_Chay" THEN "1400_KCK01_Status" := 0; END_IF;
END_REGION

REGION Network 43: Cập nhật mã trạng thái cho 1400_FT102_Status = 1 (Chạy/Mở)
   RUNG wire#powerrail
      Contact( "1400_FT102_Mo" )
      { S7_GenerateENO := "TRUE" } Move(in := 1, out1 => "1400_FT102_Status")
   END_RUNG
   // the same network as SCL:
   IF "1400_FT102_Mo" THEN "1400_FT102_Status" := 1; END_IF;
END_REGION

REGION Network 44: Cập nhật mã trạng thái cho 1400_FT102_Status = 0 (Dừng/Đóng)
   RUNG wire#powerrail
      I_Contact( "1400_FT102_Mo" )
      { S7_GenerateENO := "TRUE" } Move(in := 0, out1 => "1400_FT102_Status")
   END_RUNG
   // the same network as SCL:
   IF NOT "1400_FT102_Mo" THEN "1400_FT102_Status" := 0; END_IF;
END_REGION

REGION Network 45: Cập nhật mã trạng thái cho 1400_TY33_Status = 1 (Chạy/Mở)
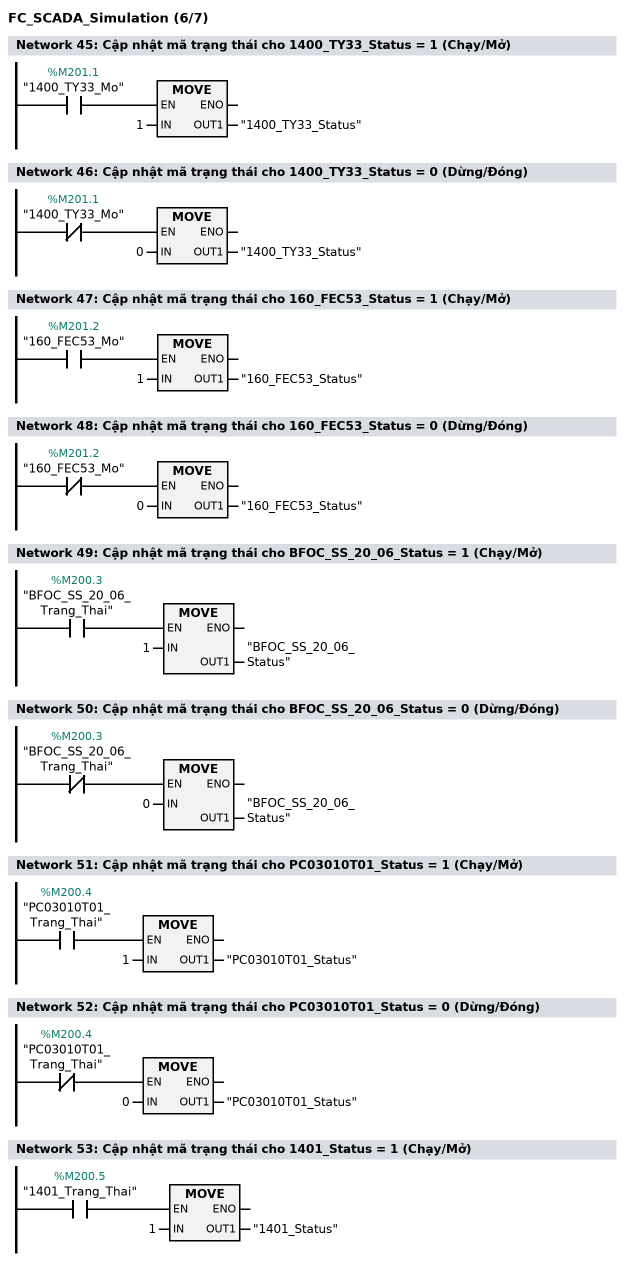
   RUNG wire#powerrail
      Contact( "1400_TY33_Mo" )
      { S7_GenerateENO := "TRUE" } Move(in := 1, out1 => "1400_TY33_Status")
   END_RUNG
   // the same network as SCL:
   IF "1400_TY33_Mo" THEN "1400_TY33_Status" := 1; END_IF;
END_REGION

REGION Network 46: Cập nhật mã trạng thái cho 1400_TY33_Status = 0 (Dừng/Đóng)
   RUNG wire#powerrail
      I_Contact( "1400_TY33_Mo" )
      { S7_GenerateENO := "TRUE" } Move(in := 0, out1 => "1400_TY33_Status")
   END_RUNG
   // the same network as SCL:
   IF NOT "1400_TY33_Mo" THEN "1400_TY33_Status" := 0; END_IF;
END_REGION

REGION Network 47: Cập nhật mã trạng thái cho 160_FEC53_Status = 1 (Chạy/Mở)
   RUNG wire#powerrail
      Contact( "160_FEC53_Mo" )
      { S7_GenerateENO := "TRUE" } Move(in := 1, out1 => "160_FEC53_Status")
   END_RUNG
   // the same network as SCL:
   IF "160_FEC53_Mo" THEN "160_FEC53_Status" := 1; END_IF;
END_REGION

REGION Network 48: Cập nhật mã trạng thái cho 160_FEC53_Status = 0 (Dừng/Đóng)
   RUNG wire#powerrail
      I_Contact( "160_FEC53_Mo" )
      { S7_GenerateENO := "TRUE" } Move(in := 0, out1 => "160_FEC53_Status")
   END_RUNG
   // the same network as SCL:
   IF NOT "160_FEC53_Mo" THEN "160_FEC53_Status" := 0; END_IF;
END_REGION

REGION Network 49: Cập nhật mã trạng thái cho BFOC_SS_20_06_Status = 1 (Chạy/Mở)
   RUNG wire#powerrail
      Contact( "BFOC_SS_20_06_Trang_Thai" )
      { S7_GenerateENO := "TRUE" } Move(in := 1, out1 => "BFOC_SS_20_06_Status")
   END_RUNG
   // the same network as SCL:
   IF "BFOC_SS_20_06_Trang_Thai" THEN "BFOC_SS_20_06_Status" := 1; END_IF;
END_REGION

REGION Network 50: Cập nhật mã trạng thái cho BFOC_SS_20_06_Status = 0 (Dừng/Đóng)
   RUNG wire#powerrail
      I_Contact( "BFOC_SS_20_06_Trang_Thai" )
      { S7_GenerateENO := "TRUE" } Move(in := 0, out1 => "BFOC_SS_20_06_Status")
   END_RUNG
   // the same network as SCL:
   IF NOT "BFOC_SS_20_06_Trang_Thai" THEN "BFOC_SS_20_06_Status" := 0; END_IF;
END_REGION

REGION Network 51: Cập nhật mã trạng thái cho PC03010T01_Status = 1 (Chạy/Mở)
   RUNG wire#powerrail
      Contact( "PC03010T01_Trang_Thai" )
      { S7_GenerateENO := "TRUE" } Move(in := 1, out1 => "PC03010T01_Status")
   END_RUNG
   // the same network as SCL:
   IF "PC03010T01_Trang_Thai" THEN "PC03010T01_Status" := 1; END_IF;
END_REGION

REGION Network 52: Cập nhật mã trạng thái cho PC03010T01_Status = 0 (Dừng/Đóng)
   RUNG wire#powerrail
      I_Contact( "PC03010T01_Trang_Thai" )
      { S7_GenerateENO := "TRUE" } Move(in := 0, out1 => "PC03010T01_Status")
   END_RUNG
   // the same network as SCL:
   IF NOT "PC03010T01_Trang_Thai" THEN "PC03010T01_Status" := 0; END_IF;
END_REGION

REGION Network 53: Cập nhật mã trạng thái cho 1401_Status = 1 (Chạy/Mở)
   RUNG wire#powerrail
      Contact( "1401_Trang_Thai" )
      { S7_GenerateENO := "TRUE" } Move(in := 1, out1 => "1401_Status")
   END_RUNG
   // the same network as SCL:
   IF "1401_Trang_Thai" THEN "1401_Status" := 1; END_IF;
END_REGION

REGION Network 54: Cập nhật mã trạng thái cho 1401_Status = 0 (Dừng/Đóng)
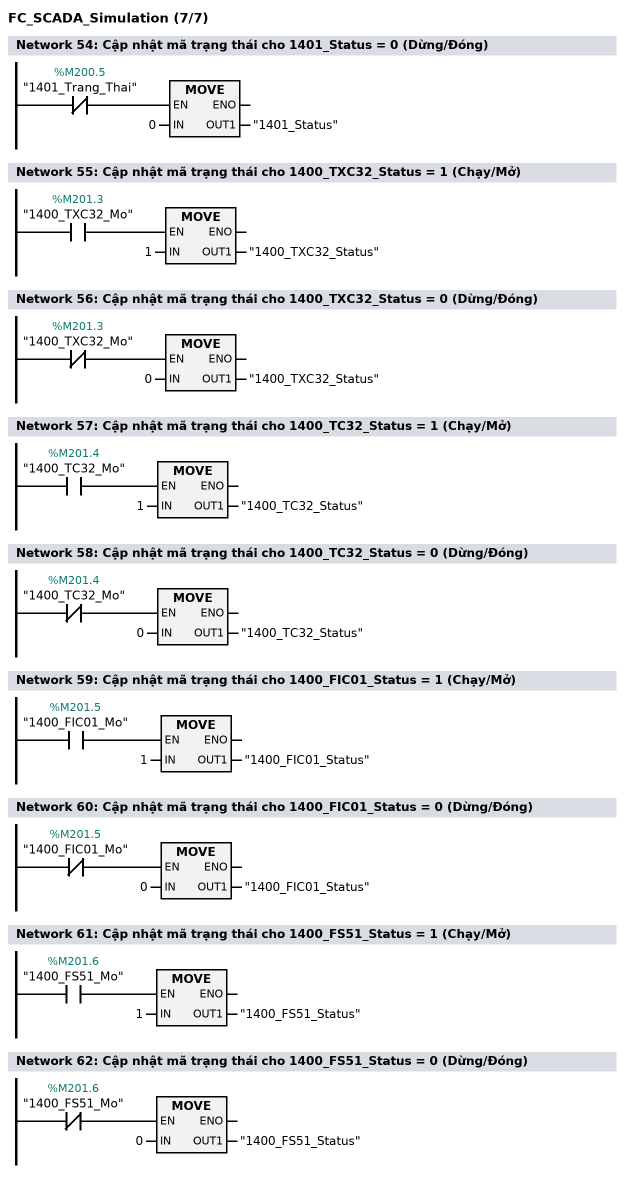
   RUNG wire#powerrail
      I_Contact( "1401_Trang_Thai" )
      { S7_GenerateENO := "TRUE" } Move(in := 0, out1 => "1401_Status")
   END_RUNG
   // the same network as SCL:
   IF NOT "1401_Trang_Thai" THEN "1401_Status" := 0; END_IF;
END_REGION

REGION Network 55: Cập nhật mã trạng thái cho 1400_TXC32_Status = 1 (Chạy/Mở)
   RUNG wire#powerrail
      Contact( "1400_TXC32_Mo" )
      { S7_GenerateENO := "TRUE" } Move(in := 1, out1 => "1400_TXC32_Status")
   END_RUNG
   // the same network as SCL:
   IF "1400_TXC32_Mo" THEN "1400_TXC32_Status" := 1; END_IF;
END_REGION

REGION Network 56: Cập nhật mã trạng thái cho 1400_TXC32_Status = 0 (Dừng/Đóng)
   RUNG wire#powerrail
      I_Contact( "1400_TXC32_Mo" )
      { S7_GenerateENO := "TRUE" } Move(in := 0, out1 => "1400_TXC32_Status")
   END_RUNG
   // the same network as SCL:
   IF NOT "1400_TXC32_Mo" THEN "1400_TXC32_Status" := 0; END_IF;
END_REGION

REGION Network 57: Cập nhật mã trạng thái cho 1400_TC32_Status = 1 (Chạy/Mở)
   RUNG wire#powerrail
      Contact( "1400_TC32_Mo" )
      { S7_GenerateENO := "TRUE" } Move(in := 1, out1 => "1400_TC32_Status")
   END_RUNG
   // the same network as SCL:
   IF "1400_TC32_Mo" THEN "1400_TC32_Status" := 1; END_IF;
END_REGION

REGION Network 58: Cập nhật mã trạng thái cho 1400_TC32_Status = 0 (Dừng/Đóng)
   RUNG wire#powerrail
      I_Contact( "1400_TC32_Mo" )
      { S7_GenerateENO := "TRUE" } Move(in := 0, out1 => "1400_TC32_Status")
   END_RUNG
   // the same network as SCL:
   IF NOT "1400_TC32_Mo" THEN "1400_TC32_Status" := 0; END_IF;
END_REGION

REGION Network 59: Cập nhật mã trạng thái cho 1400_FIC01_Status = 1 (Chạy/Mở)
   RUNG wire#powerrail
      Contact( "1400_FIC01_Mo" )
      { S7_GenerateENO := "TRUE" } Move(in := 1, out1 => "1400_FIC01_Status")
   END_RUNG
   // the same network as SCL:
   IF "1400_FIC01_Mo" THEN "1400_FIC01_Status" := 1; END_IF;
END_REGION

REGION Network 60: Cập nhật mã trạng thái cho 1400_FIC01_Status = 0 (Dừng/Đóng)
   RUNG wire#powerrail
      I_Contact( "1400_FIC01_Mo" )
      { S7_GenerateENO := "TRUE" } Move(in := 0, out1 => "1400_FIC01_Status")
   END_RUNG
   // the same network as SCL:
   IF NOT "1400_FIC01_Mo" THEN "1400_FIC01_Status" := 0; END_IF;
END_REGION

REGION Network 61: Cập nhật mã trạng thái cho 1400_FS51_Status = 1 (Chạy/Mở)
   RUNG wire#powerrail
      Contact( "1400_FS51_Mo" )
      { S7_GenerateENO := "TRUE" } Move(in := 1, out1 => "1400_FS51_Status")
   END_RUNG
   // the same network as SCL:
   IF "1400_FS51_Mo" THEN "1400_FS51_Status" := 1; END_IF;
END_REGION

REGION Network 62: Cập nhật mã trạng thái cho 1400_FS51_Status = 0 (Dừng/Đóng)
   RUNG wire#powerrail
      I_Contact( "1400_FS51_Mo" )
      { S7_GenerateENO := "TRUE" } Move(in := 0, out1 => "1400_FS51_Status")
   END_RUNG
   // the same network as SCL:
   IF NOT "1400_FS51_Mo" THEN "1400_FS51_Status" := 0; END_IF;
END_REGION
END_FUNCTION

BLOCK "WT_Temp_Schema"   // PlcWatchTable
BEGIN
END_BLOCK

BLOCK "WT_Test_Import_DB_Schema"   // PlcWatchTable
BEGIN
END_BLOCK

BLOCK "WT_Test_Import_Schema"   // PlcWatchTable
BEGIN
END_BLOCK

FUNCTION_BLOCK "A_COUNTER"   // FB12, LAD
VERSION : 0.1
// stored: AutoNumber true, IsIECCheckEnabled false, UDAEnableTagReadback false
BEGIN

REGION Network 1
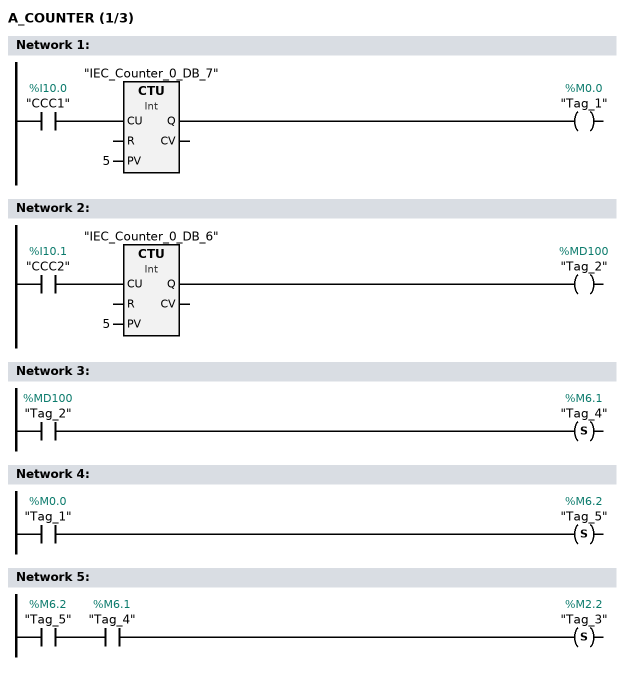
   RUNG wire#powerrail
      Contact( "CCC1" )
      { S7_Templates := "value_type := Int" } "IEC_Counter_0_DB_7".CTU(r :=, pv := 5, cv =>)
      Coil( "Tag_1" )
   END_RUNG
   // the same network as SCL:
   "IEC_Counter_0_DB_7".CTU(CU := "CCC1", PV := 5);
   "Tag_1" := "IEC_Counter_0_DB_7".Q;
END_REGION

REGION Network 2
   RUNG wire#powerrail
      Contact( "CCC2" )
      { S7_Templates := "value_type := Int" } "IEC_Counter_0_DB_6".CTU(r :=, pv := 5, cv =>)
      Coil( "Tag_2" )
   END_RUNG
   // the same network as SCL:
   "IEC_Counter_0_DB_6".CTU(CU := "CCC2", PV := 5);
   "Tag_2" := "IEC_Counter_0_DB_6".Q;
END_REGION

REGION Network 3
   RUNG wire#powerrail
      Contact( "Tag_2" )
      S_Coil( "Tag_4" )
   END_RUNG
   // the same network as SCL:
   IF "Tag_2" THEN "Tag_4" := TRUE; END_IF;
END_REGION

REGION Network 4
   RUNG wire#powerrail
      Contact( "Tag_1" )
      S_Coil( "Tag_5" )
   END_RUNG
   // the same network as SCL:
   IF "Tag_1" THEN "Tag_5" := TRUE; END_IF;
END_REGION

REGION Network 5
   RUNG wire#powerrail
      Contact( "Tag_5" )
      Contact( "Tag_4" )
      S_Coil( "Tag_3" )
   END_RUNG
   // the same network as SCL:
   IF "Tag_5" AND "Tag_4" THEN "Tag_3" := TRUE; END_IF;
END_REGION

REGION Network 6
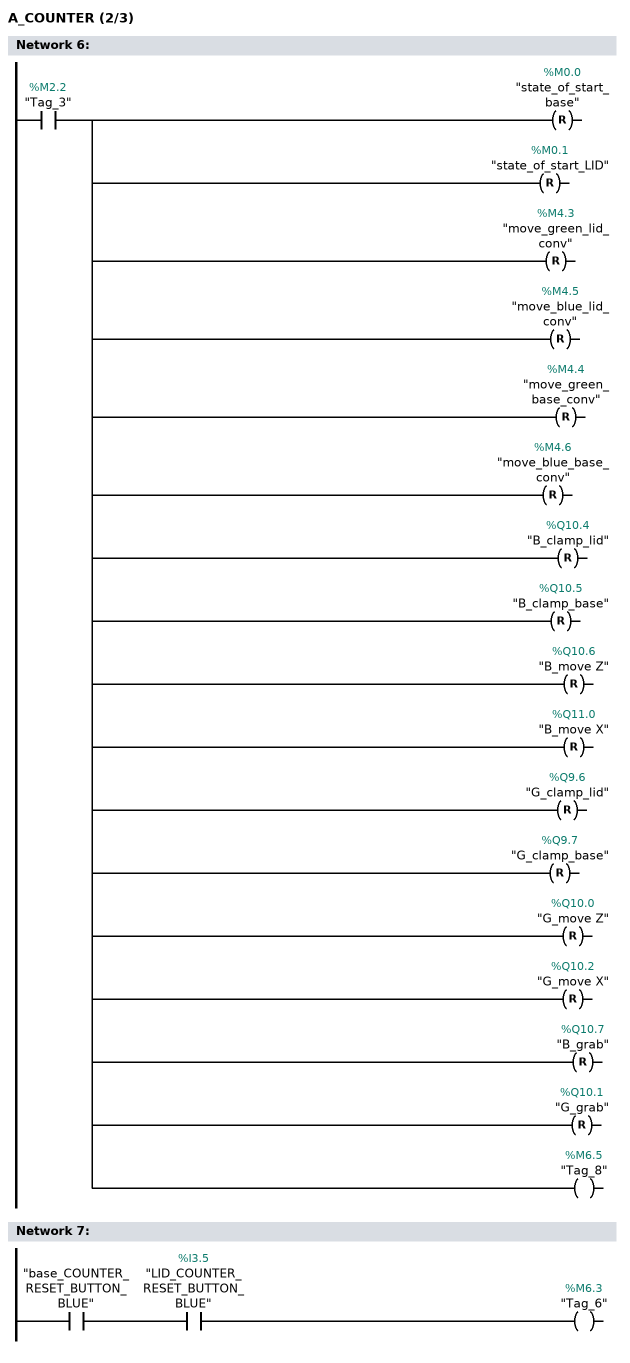
   RUNG wire#powerrail
      Contact( "Tag_3" )
      wire#w1
      R_Coil( "state_of_start_base" )
   END_RUNG
   RUNG wire#w1
      R_Coil( "state_of_start_LID" )
   END_RUNG
   RUNG wire#w1
      R_Coil( "move_green_lid_conv" )
   END_RUNG
   RUNG wire#w1
      R_Coil( "move_blue_lid_conv" )
   END_RUNG
   RUNG wire#w1
      R_Coil( "move_green_base_conv" )
   END_RUNG
   RUNG wire#w1
      R_Coil( "move_blue_base_conv" )
   END_RUNG
   RUNG wire#w1
      R_Coil( "B_clamp_lid" )
   END_RUNG
   RUNG wire#w1
      R_Coil( "B_clamp_base" )
   END_RUNG
   RUNG wire#w1
      R_Coil( "B_move Z" )
   END_RUNG
   RUNG wire#w1
      R_Coil( "B_move X" )
   END_RUNG
   RUNG wire#w1
      R_Coil( "G_clamp_lid" )
   END_RUNG
   RUNG wire#w1
      R_Coil( "G_clamp_base" )
   END_RUNG
   RUNG wire#w1
      R_Coil( "G_move Z" )
   END_RUNG
   RUNG wire#w1
      R_Coil( "G_move X" )
   END_RUNG
   RUNG wire#w1
      R_Coil( "B_grab" )
   END_RUNG
   RUNG wire#w1
      R_Coil( "G_grab" )
   END_RUNG
   RUNG wire#w1
      Coil( "Tag_8" )
   END_RUNG
   // the same network as SCL:
   IF "Tag_3" THEN
       "state_of_start_base" := FALSE;
       "state_of_start_LID" := FALSE;
       "move_green_lid_conv" := FALSE;
       "move_blue_lid_conv" := FALSE;
       "move_green_base_conv" := FALSE;
       "move_blue_base_conv" := FALSE;
       "B_clamp_lid" := FALSE;
       "B_clamp_base" := FALSE;
       "B_move Z" := FALSE;
       "B_move X" := FALSE;
       "G_clamp_lid" := FALSE;
       "G_clamp_base" := FALSE;
       "G_move Z" := FALSE;
       "G_move X" := FALSE;
       "B_grab" := FALSE;
       "G_grab" := FALSE;
   END_IF;
   "Tag_8" := "Tag_3";
END_REGION

REGION Network 7
   RUNG wire#powerrail
      Contact( "base_COUNTER_RESET_BUTTON_BLUE" )
      Contact( "LID_COUNTER_RESET_BUTTON_BLUE" )
      Coil( "Tag_6" )
   END_RUNG
   // the same network as SCL:
   "Tag_6" := "base_COUNTER_RESET_BUTTON_BLUE" AND "LID_COUNTER_RESET_BUTTON_BLUE";
END_REGION

REGION Network 8
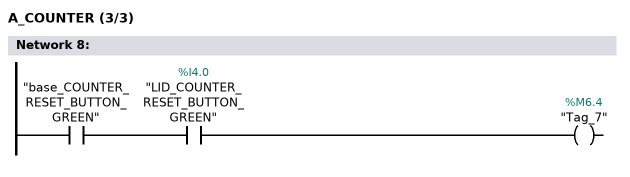
   RUNG wire#powerrail
      Contact( "base_COUNTER_RESET_BUTTON_GREEN" )
      Contact( "LID_COUNTER_RESET_BUTTON_GREEN" )
      Coil( "Tag_7" )
   END_RUNG
   // the same network as SCL:
   "Tag_7" := "base_COUNTER_RESET_BUTTON_GREEN" AND "LID_COUNTER_RESET_BUTTON_GREEN";
END_REGION
END_FUNCTION_BLOCK

FUNCTION_BLOCK "Assembly_conv"   // FB9, LAD
VERSION : 0.1
// stored: AutoNumber true, IsIECCheckEnabled false, UDAEnableTagReadback false
   VAR_TEMP   // added for the SCL form of the ladder/FBD networks
      _w1 : Bool;
      _s5time1 : S5Time;
   END_VAR
BEGIN

REGION Network 1
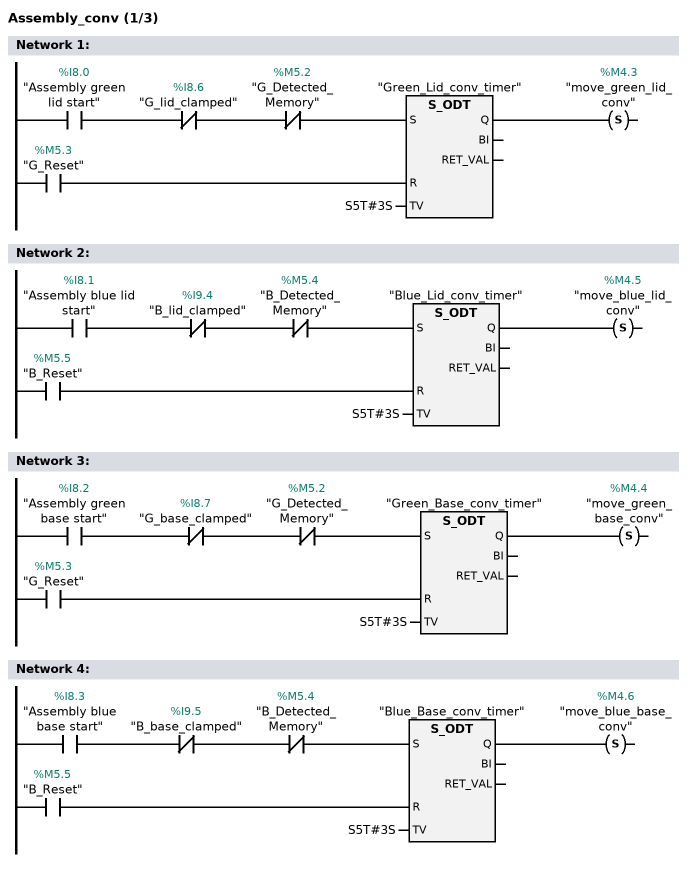
   RUNG wire#powerrail
      Contact( "Assembly green lid start" )
      I_Contact( "G_lid_clamped" )
      I_Contact( "G_Detected_Memory" )
      S_ODT(T_NO := "Green_Lid_conv_timer", R := wire#w1, TV := S5T#3S, BI =>, RET_VAL =>)
      S_Coil( "move_green_lid_conv" )
   END_RUNG
   RUNG wire#powerrail
      Contact( "G_Reset" )
   END_RUNG wire#w1
   // the same network as SCL:
   #_s5time1 := S_ODT(T_NO := "Green_Lid_conv_timer",
                      S := "Assembly green lid start" AND NOT "G_lid_clamped" AND NOT "G_Detected_Memory",
                      R := "G_Reset",
                      TV := S5T#3S,
                      Q => #_w1);
   IF #_w1 THEN "move_green_lid_conv" := TRUE; END_IF;
END_REGION

REGION Network 2
   RUNG wire#powerrail
      Contact( "Assembly blue lid start" )
      I_Contact( "B_lid_clamped" )
      I_Contact( "B_Detected_Memory" )
      S_ODT(T_NO := "Blue_Lid_conv_timer", R := wire#w1, TV := S5T#3S, BI =>, RET_VAL =>)
      S_Coil( "move_blue_lid_conv" )
   END_RUNG
   RUNG wire#powerrail
      Contact( "B_Reset" )
   END_RUNG wire#w1
   // the same network as SCL:
   #_s5time1 := S_ODT(T_NO := "Blue_Lid_conv_timer",
                      S := "Assembly blue lid start" AND NOT "B_lid_clamped" AND NOT "B_Detected_Memory",
                      R := "B_Reset",
                      TV := S5T#3S,
                      Q => #_w1);
   IF #_w1 THEN "move_blue_lid_conv" := TRUE; END_IF;
END_REGION

REGION Network 3
   RUNG wire#powerrail
      Contact( "Assembly green base start" )
      I_Contact( "G_base_clamped" )
      I_Contact( "G_Detected_Memory" )
      S_ODT(T_NO := "Green_Base_conv_timer", R := wire#w1, TV := S5T#3S, BI =>, RET_VAL =>)
      S_Coil( "move_green_base_conv" )
   END_RUNG
   RUNG wire#powerrail
      Contact( "G_Reset" )
   END_RUNG wire#w1
   // the same network as SCL:
   #_s5time1 := S_ODT(T_NO := "Green_Base_conv_timer",
                      S := "Assembly green base start" AND NOT "G_base_clamped" AND NOT "G_Detected_Memory",
                      R := "G_Reset",
                      TV := S5T#3S,
                      Q => #_w1);
   IF #_w1 THEN "move_green_base_conv" := TRUE; END_IF;
END_REGION

REGION Network 4
   RUNG wire#powerrail
      Contact( "Assembly blue base start" )
      I_Contact( "B_base_clamped" )
      I_Contact( "B_Detected_Memory" )
      S_ODT(T_NO := "Blue_Base_conv_timer", R := wire#w1, TV := S5T#3S, BI =>, RET_VAL =>)
      S_Coil( "move_blue_base_conv" )
   END_RUNG
   RUNG wire#powerrail
      Contact( "B_Reset" )
   END_RUNG wire#w1
   // the same network as SCL:
   #_s5time1 := S_ODT(T_NO := "Blue_Base_conv_timer",
                      S := "Assembly blue base start" AND NOT "B_base_clamped" AND NOT "B_Detected_Memory",
                      R := "B_Reset",
                      TV := S5T#3S,
                      Q => #_w1);
   IF #_w1 THEN "move_blue_base_conv" := TRUE; END_IF;
END_REGION

REGION Network 5
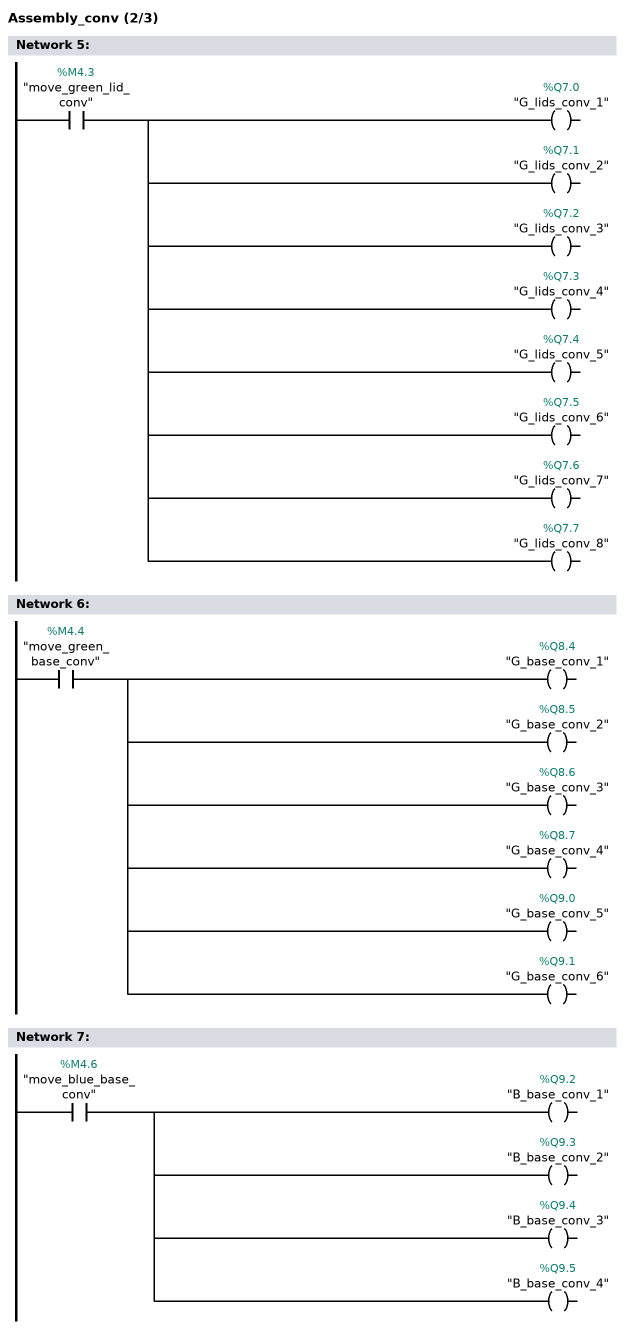
   RUNG wire#powerrail
      Contact( "move_green_lid_conv" )
      wire#w1
      Coil( "G_lids_conv_1" )
   END_RUNG
   RUNG wire#w1
      Coil( "G_lids_conv_2" )
   END_RUNG
   RUNG wire#w1
      Coil( "G_lids_conv_3" )
   END_RUNG
   RUNG wire#w1
      Coil( "G_lids_conv_4" )
   END_RUNG
   RUNG wire#w1
      Coil( "G_lids_conv_5" )
   END_RUNG
   RUNG wire#w1
      Coil( "G_lids_conv_6" )
   END_RUNG
   RUNG wire#w1
      Coil( "G_lids_conv_7" )
   END_RUNG
   RUNG wire#w1
      Coil( "G_lids_conv_8" )
   END_RUNG
   // the same network as SCL:
   "G_lids_conv_1" := "move_green_lid_conv";
   "G_lids_conv_2" := "move_green_lid_conv";
   "G_lids_conv_3" := "move_green_lid_conv";
   "G_lids_conv_4" := "move_green_lid_conv";
   "G_lids_conv_5" := "move_green_lid_conv";
   "G_lids_conv_6" := "move_green_lid_conv";
   "G_lids_conv_7" := "move_green_lid_conv";
   "G_lids_conv_8" := "move_green_lid_conv";
END_REGION

REGION Network 6
   RUNG wire#powerrail
      Contact( "move_green_base_conv" )
      wire#w1
      Coil( "G_base_conv_1" )
   END_RUNG
   RUNG wire#w1
      Coil( "G_base_conv_2" )
   END_RUNG
   RUNG wire#w1
      Coil( "G_base_conv_3" )
   END_RUNG
   RUNG wire#w1
      Coil( "G_base_conv_4" )
   END_RUNG
   RUNG wire#w1
      Coil( "G_base_conv_5" )
   END_RUNG
   RUNG wire#w1
      Coil( "G_base_conv_6" )
   END_RUNG
   // the same network as SCL:
   "G_base_conv_1" := "move_green_base_conv";
   "G_base_conv_2" := "move_green_base_conv";
   "G_base_conv_3" := "move_green_base_conv";
   "G_base_conv_4" := "move_green_base_conv";
   "G_base_conv_5" := "move_green_base_conv";
   "G_base_conv_6" := "move_green_base_conv";
END_REGION

REGION Network 7
   RUNG wire#powerrail
      Contact( "move_blue_base_conv" )
      wire#w1
      Coil( "B_base_conv_1" )
   END_RUNG
   RUNG wire#w1
      Coil( "B_base_conv_2" )
   END_RUNG
   RUNG wire#w1
      Coil( "B_base_conv_3" )
   END_RUNG
   RUNG wire#w1
      Coil( "B_base_conv_4" )
   END_RUNG
   // the same network as SCL:
   "B_base_conv_1" := "move_blue_base_conv";
   "B_base_conv_2" := "move_blue_base_conv";
   "B_base_conv_3" := "move_blue_base_conv";
   "B_base_conv_4" := "move_blue_base_conv";
END_REGION

REGION Network 8
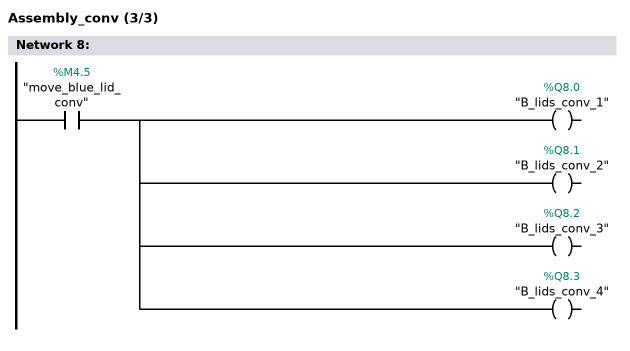
   RUNG wire#powerrail
      Contact( "move_blue_lid_conv" )
      wire#w1
      Coil( "B_lids_conv_1" )
   END_RUNG
   RUNG wire#w1
      Coil( "B_lids_conv_2" )
   END_RUNG
   RUNG wire#w1
      Coil( "B_lids_conv_3" )
   END_RUNG
   RUNG wire#w1
      Coil( "B_lids_conv_4" )
   END_RUNG
   // the same network as SCL:
   "B_lids_conv_1" := "move_blue_lid_conv";
   "B_lids_conv_2" := "move_blue_lid_conv";
   "B_lids_conv_3" := "move_blue_lid_conv";
   "B_lids_conv_4" := "move_blue_lid_conv";
END_REGION
END_FUNCTION_BLOCK

FUNCTION_BLOCK "BASE_execess_remove_station"   // FB7, LAD
VERSION : 0.1
// stored: AutoNumber true, IsIECCheckEnabled false, UDAEnableTagReadback false
BEGIN

REGION Network 1: LID_BELT_EXECESS_CONVYR_HANDLER
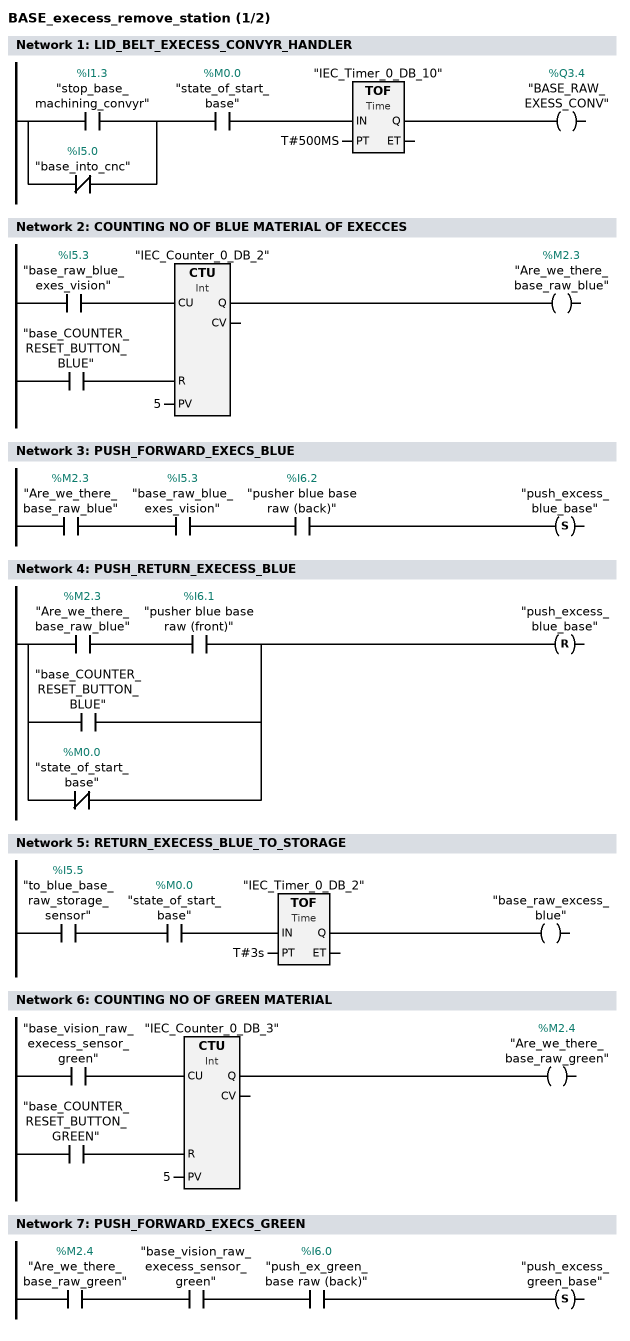
   RUNG wire#powerrail
      Contact( "stop_base_machining_convyr" )
      wire#w1
      Contact( "state_of_start_base" )
      { S7_Templates := "time_type := Time" } "IEC_Timer_0_DB_10".TOF(pt := T#500MS, et =>)
      Coil( "BASE_RAW_EXESS_CONV" )
   END_RUNG
   RUNG wire#powerrail
      I_Contact( "base_into_cnc" )
   END_RUNG wire#w1
   // the same network as SCL:
   "IEC_Timer_0_DB_10".TOF(IN := ("stop_base_machining_convyr" OR NOT "base_into_cnc") AND "state_of_start_base",
                           PT := T#500MS);
   "BASE_RAW_EXESS_CONV" := "IEC_Timer_0_DB_10".Q;
END_REGION

REGION Network 2: COUNTING NO OF BLUE MATERIAL OF EXECCES
   RUNG wire#powerrail
      Contact( "base_raw_blue_exes_vision" )
      { S7_Templates := "value_type := Int" } "IEC_Counter_0_DB_2".CTU(r := wire#w1, pv := 5, cv =>)
      Coil( "Are_we_there_base_raw_blue" )
   END_RUNG
   RUNG wire#powerrail
      Contact( "base_COUNTER_RESET_BUTTON_BLUE" )
   END_RUNG wire#w1
   // the same network as SCL:
   "IEC_Counter_0_DB_2".CTU(CU := "base_raw_blue_exes_vision", R := "base_COUNTER_RESET_BUTTON_BLUE", PV := 5);
   "Are_we_there_base_raw_blue" := "IEC_Counter_0_DB_2".Q;
END_REGION

REGION Network 3: PUSH_FORWARD_EXECS_BLUE
   RUNG wire#powerrail
      Contact( "Are_we_there_base_raw_blue" )
      Contact( "base_raw_blue_exes_vision" )
      Contact( "pusher blue base raw (back)" )
      S_Coil( "push_excess_blue_base" )
   END_RUNG
   // the same network as SCL:
   IF "Are_we_there_base_raw_blue" AND "base_raw_blue_exes_vision" AND "pusher blue base raw (back)" THEN
       "push_excess_blue_base" := TRUE;
   END_IF;
END_REGION

REGION Network 4: PUSH_RETURN_EXECESS_BLUE
   RUNG wire#powerrail
      Contact( "Are_we_there_base_raw_blue" )
      Contact( "pusher blue base raw (front)" )
      wire#w1
      R_Coil( "push_excess_blue_base" )
   END_RUNG
   RUNG wire#powerrail
      Contact( "base_COUNTER_RESET_BUTTON_BLUE" )
   END_RUNG wire#w1
   RUNG wire#powerrail
      I_Contact( "state_of_start_base" )
   END_RUNG wire#w1
   // the same network as SCL:
   IF ("Are_we_there_base_raw_blue" AND "pusher blue base raw (front)") OR "base_COUNTER_RESET_BUTTON_BLUE" OR NOT "state_of_start_base" THEN
       "push_excess_blue_base" := FALSE;
   END_IF;
END_REGION

REGION Network 5: RETURN_EXECESS_BLUE_TO_STORAGE
   RUNG wire#powerrail
      Contact( "to_blue_base_raw_storage_sensor" )
      Contact( "state_of_start_base" )
      { S7_Templates := "time_type := Time" } "IEC_Timer_0_DB_2".TOF(pt := T#3s, et =>)
      Coil( "base_raw_excess_blue" )
   END_RUNG
   // the same network as SCL:
   "IEC_Timer_0_DB_2".TOF(IN := "to_blue_base_raw_storage_sensor" AND "state_of_start_base", PT := T#3s);
   "base_raw_excess_blue" := "IEC_Timer_0_DB_2".Q;
END_REGION

REGION Network 6: COUNTING NO OF GREEN MATERIAL
   RUNG wire#powerrail
      Contact( "base_vision_raw_execess_sensor_green" )
      { S7_Templates := "value_type := Int" } "IEC_Counter_0_DB_3".CTU(r := wire#w1, pv := 5, cv =>)
      Coil( "Are_we_there_base_raw_green" )
   END_RUNG
   RUNG wire#powerrail
      Contact( "base_COUNTER_RESET_BUTTON_GREEN" )
   END_RUNG wire#w1
   // the same network as SCL:
   "IEC_Counter_0_DB_3".CTU(CU := "base_vision_raw_execess_sensor_green",
                           R := "base_COUNTER_RESET_BUTTON_GREEN",
                           PV := 5);
   "Are_we_there_base_raw_green" := "IEC_Counter_0_DB_3".Q;
END_REGION

REGION Network 7: PUSH_FORWARD_EXECS_GREEN
   RUNG wire#powerrail
      Contact( "Are_we_there_base_raw_green" )
      Contact( "base_vision_raw_execess_sensor_green" )
      Contact( "push_ex_green_base raw (back)" )
      S_Coil( "push_excess_green_base" )
   END_RUNG
   // the same network as SCL:
   IF "Are_we_there_base_raw_green" AND "base_vision_raw_execess_sensor_green" AND "push_ex_green_base raw (back)" THEN
       "push_excess_green_base" := TRUE;
   END_IF;
END_REGION

REGION Network 8: RETURN_EXECESS_GREEN_TO_STORAGE
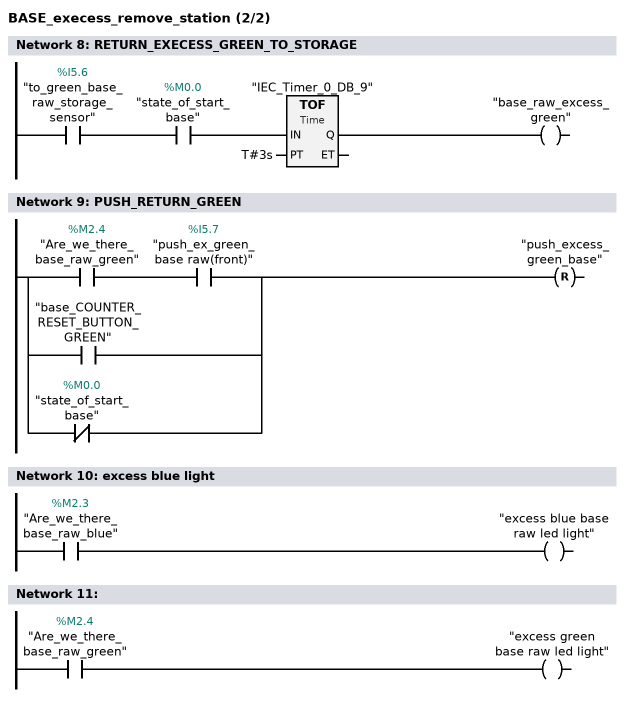
   RUNG wire#powerrail
      Contact( "to_green_base_raw_storage_sensor" )
      Contact( "state_of_start_base" )
      { S7_Templates := "time_type := Time" } "IEC_Timer_0_DB_9".TOF(pt := T#3s, et =>)
      Coil( "base_raw_excess_green" )
   END_RUNG
   // the same network as SCL:
   "IEC_Timer_0_DB_9".TOF(IN := "to_green_base_raw_storage_sensor" AND "state_of_start_base", PT := T#3s);
   "base_raw_excess_green" := "IEC_Timer_0_DB_9".Q;
END_REGION

REGION Network 9: PUSH_RETURN_GREEN
   RUNG wire#powerrail
      Contact( "Are_we_there_base_raw_green" )
      Contact( "push_ex_green_base raw(front)" )
      wire#w1
      R_Coil( "push_excess_green_base" )
   END_RUNG
   RUNG wire#powerrail
      Contact( "base_COUNTER_RESET_BUTTON_GREEN" )
   END_RUNG wire#w1
   RUNG wire#powerrail
      I_Contact( "state_of_start_base" )
   END_RUNG wire#w1
   // the same network as SCL:
   IF ("Are_we_there_base_raw_green" AND "push_ex_green_base raw(front)") OR "base_COUNTER_RESET_BUTTON_GREEN" OR NOT "state_of_start_base" THEN
       "push_excess_green_base" := FALSE;
   END_IF;
END_REGION

REGION Network 10: excess blue light
   RUNG wire#powerrail
      Contact( "Are_we_there_base_raw_blue" )
      Coil( "excess blue base raw led light" )
   END_RUNG
   // the same network as SCL:
   "excess blue base raw led light" := "Are_we_there_base_raw_blue";
END_REGION

REGION Network 11
   RUNG wire#powerrail
      Contact( "Are_we_there_base_raw_green" )
      Coil( "excess green base raw led light" )
   END_RUNG
   // the same network as SCL:
   "excess green base raw led light" := "Are_we_there_base_raw_green";
END_REGION
END_FUNCTION_BLOCK

FUNCTION "FC_AUTO_MODE" : Void   // FC2, LAD
{ S7_Optimized_Access := 'TRUE' }
VERSION : 0.1
// stored: AutoNumber true, IsIECCheckEnabled false, SetENOAutomatically false, UDAEnableTagReadback false
   VAR_TEMP   // added for the SCL form of the ladder/FBD networks
      _w1 : Bool;
      _w2 : Bool;
      _w3 : Bool;
      _w4 : Bool;
      _w5 : Bool;
      _w6 : Bool;
   END_VAR
BEGIN

REGION Network 1: RESET CÁC BỘ ĐẾM VỀ 0
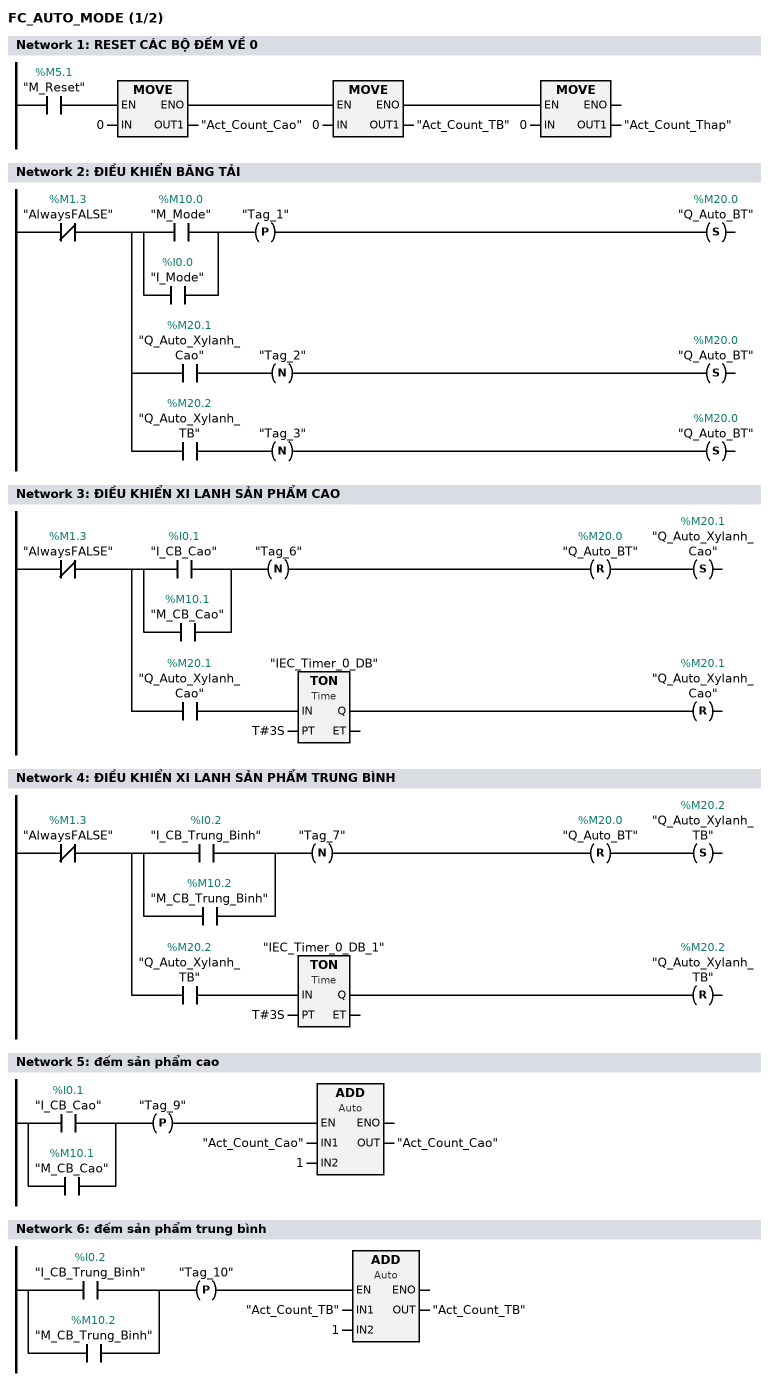
   RUNG wire#powerrail
      Contact( "M_Reset" )
      Move(in := 0, out1 => "Act_Count_Cao")
      Move(in := 0, out1 => "Act_Count_TB")
      Move(in := 0, out1 => "Act_Count_Thap")
   END_RUNG
   // the same network as SCL:
   IF "M_Reset" THEN
       "Act_Count_Cao" := 0;
       "Act_Count_TB" := 0;
       "Act_Count_Thap" := 0;
   END_IF;
END_REGION

REGION Network 2: ĐIỀU KHIỂN BĂNG TẢI
   RUNG wire#powerrail
      I_Contact( "AlwaysFALSE" )
      wire#w1
      Contact( "M_Mode" )
      wire#w2
      P_Trig( "Tag_1" )
      S_Coil( "Q_Auto_BT" )
   END_RUNG
   RUNG wire#w1
      Contact( "I_Mode" )
   END_RUNG wire#w2
   RUNG wire#w1
      Contact( "Q_Auto_Xylanh_Cao" )
      N_Trig( "Tag_2" )
      S_Coil( "Q_Auto_BT" )
   END_RUNG
   RUNG wire#w1
      Contact( "Q_Auto_Xylanh_TB" )
      N_Trig( "Tag_3" )
      S_Coil( "Q_Auto_BT" )
   END_RUNG
   // the same network as SCL:
   #_w1 := NOT "AlwaysFALSE" AND ("M_Mode" OR "I_Mode");
   #_w2 := #_w1 AND NOT "Tag_1";   // rising edge
   "Tag_1" := #_w1;
   IF #_w2 THEN "Q_Auto_BT" := TRUE; END_IF;
   #_w3 := NOT "AlwaysFALSE" AND "Q_Auto_Xylanh_Cao";
   #_w4 := NOT #_w3 AND "Tag_2";   // falling edge
   "Tag_2" := #_w3;
   IF #_w4 THEN "Q_Auto_BT" := TRUE; END_IF;
   #_w5 := NOT "AlwaysFALSE" AND "Q_Auto_Xylanh_TB";
   #_w6 := NOT #_w5 AND "Tag_3";   // falling edge
   "Tag_3" := #_w5;
   IF #_w6 THEN "Q_Auto_BT" := TRUE; END_IF;
END_REGION

REGION Network 3: ĐIỀU KHIỂN XI LANH SẢN PHẨM CAO
   RUNG wire#powerrail
      I_Contact( "AlwaysFALSE" )
      wire#w1
      Contact( "I_CB_Cao" )
      wire#w2
      N_Trig( "Tag_6" )
      R_Coil( "Q_Auto_BT" )
      S_Coil( "Q_Auto_Xylanh_Cao" )
   END_RUNG
   RUNG wire#w1
      Contact( "M_CB_Cao" )
   END_RUNG wire#w2
   RUNG wire#w1
      Contact( "Q_Auto_Xylanh_Cao" )
      { S7_Templates := "time_type := Time" } "IEC_Timer_0_DB".TON(pt := T#3S, et =>)
      R_Coil( "Q_Auto_Xylanh_Cao" )
   END_RUNG
   // the same network as SCL:
   #_w1 := NOT "AlwaysFALSE" AND ("I_CB_Cao" OR "M_CB_Cao");
   #_w2 := NOT #_w1 AND "Tag_6";   // falling edge
   "Tag_6" := #_w1;
   IF #_w2 THEN
       "Q_Auto_BT" := FALSE;
       "Q_Auto_Xylanh_Cao" := TRUE;
   END_IF;
   "IEC_Timer_0_DB".TON(IN := NOT "AlwaysFALSE" AND "Q_Auto_Xylanh_Cao", PT := T#3S);
   IF "IEC_Timer_0_DB".Q THEN "Q_Auto_Xylanh_Cao" := FALSE; END_IF;
END_REGION

REGION Network 4: ĐIỀU KHIỂN XI LANH SẢN PHẨM TRUNG BÌNH
   RUNG wire#powerrail
      I_Contact( "AlwaysFALSE" )
      wire#w1
      Contact( "I_CB_Trung_Binh" )
      wire#w2
      N_Trig( "Tag_7" )
      R_Coil( "Q_Auto_BT" )
      S_Coil( "Q_Auto_Xylanh_TB" )
   END_RUNG
   RUNG wire#w1
      Contact( "M_CB_Trung_Binh" )
   END_RUNG wire#w2
   RUNG wire#w1
      Contact( "Q_Auto_Xylanh_TB" )
      { S7_Templates := "time_type := Time" } "IEC_Timer_0_DB_1".TON(pt := T#3S, et =>)
      R_Coil( "Q_Auto_Xylanh_TB" )
   END_RUNG
   // the same network as SCL:
   #_w1 := NOT "AlwaysFALSE" AND ("I_CB_Trung_Binh" OR "M_CB_Trung_Binh");
   #_w2 := NOT #_w1 AND "Tag_7";   // falling edge
   "Tag_7" := #_w1;
   IF #_w2 THEN
       "Q_Auto_BT" := FALSE;
       "Q_Auto_Xylanh_TB" := TRUE;
   END_IF;
   "IEC_Timer_0_DB_1".TON(IN := NOT "AlwaysFALSE" AND "Q_Auto_Xylanh_TB", PT := T#3S);
   IF "IEC_Timer_0_DB_1".Q THEN "Q_Auto_Xylanh_TB" := FALSE; END_IF;
END_REGION

REGION Network 5: đếm sản phẩm cao
   RUNG wire#powerrail
      Contact( "I_CB_Cao" )
      wire#w1
      P_Trig( "Tag_9" )
      Add(in1 := "Act_Count_Cao", in2 := 1, out => "Act_Count_Cao")
   END_RUNG
   RUNG wire#powerrail
      Contact( "M_CB_Cao" )
   END_RUNG wire#w1
   // the same network as SCL:
   #_w1 := "I_CB_Cao" OR "M_CB_Cao";
   #_w2 := #_w1 AND NOT "Tag_9";   // rising edge
   "Tag_9" := #_w1;
   IF #_w2 THEN "Act_Count_Cao" := "Act_Count_Cao" + 1; END_IF;
END_REGION

REGION Network 6: đếm sản phẩm trung bình
   RUNG wire#powerrail
      Contact( "I_CB_Trung_Binh" )
      wire#w1
      P_Trig( "Tag_10" )
      Add(in1 := "Act_Count_TB", in2 := 1, out => "Act_Count_TB")
   END_RUNG
   RUNG wire#powerrail
      Contact( "M_CB_Trung_Binh" )
   END_RUNG wire#w1
   // the same network as SCL:
   #_w1 := "I_CB_Trung_Binh" OR "M_CB_Trung_Binh";
   #_w2 := #_w1 AND NOT "Tag_10";   // rising edge
   "Tag_10" := #_w1;
   IF #_w2 THEN "Act_Count_TB" := "Act_Count_TB" + 1; END_IF;
END_REGION

REGION Network 7: đếm sản phẩm thấp
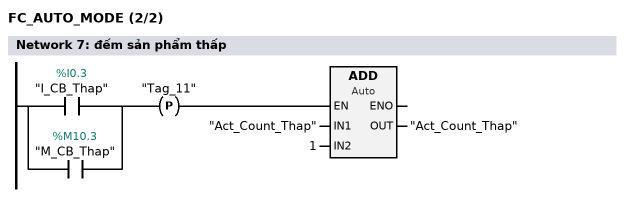
   RUNG wire#powerrail
      Contact( "I_CB_Thap" )
      wire#w1
      P_Trig( "Tag_11" )
      Add(in1 := "Act_Count_Thap", in2 := 1, out => "Act_Count_Thap")
   END_RUNG
   RUNG wire#powerrail
      Contact( "M_CB_Thap" )
   END_RUNG wire#w1
   // the same network as SCL:
   #_w1 := "I_CB_Thap" OR "M_CB_Thap";
   #_w2 := #_w1 AND NOT "Tag_11";   // rising edge
   "Tag_11" := #_w1;
   IF #_w2 THEN "Act_Count_Thap" := "Act_Count_Thap" + 1; END_IF;
END_REGION
END_FUNCTION

FUNCTION "FC_Bon_Chua_Loc" : Void   // FC30, LAD
{ S7_Optimized_Access := 'TRUE' }
VERSION : 0.1
// stored: AutoNumber true, IsIECCheckEnabled false
   VAR_TEMP   // added for the SCL form of the ladder/FBD networks
      _w1 : Bool;
   END_VAR
BEGIN

REGION Network 1: Gated HMI AI_LSH3310_Pheu_Cao qua Sim Mode
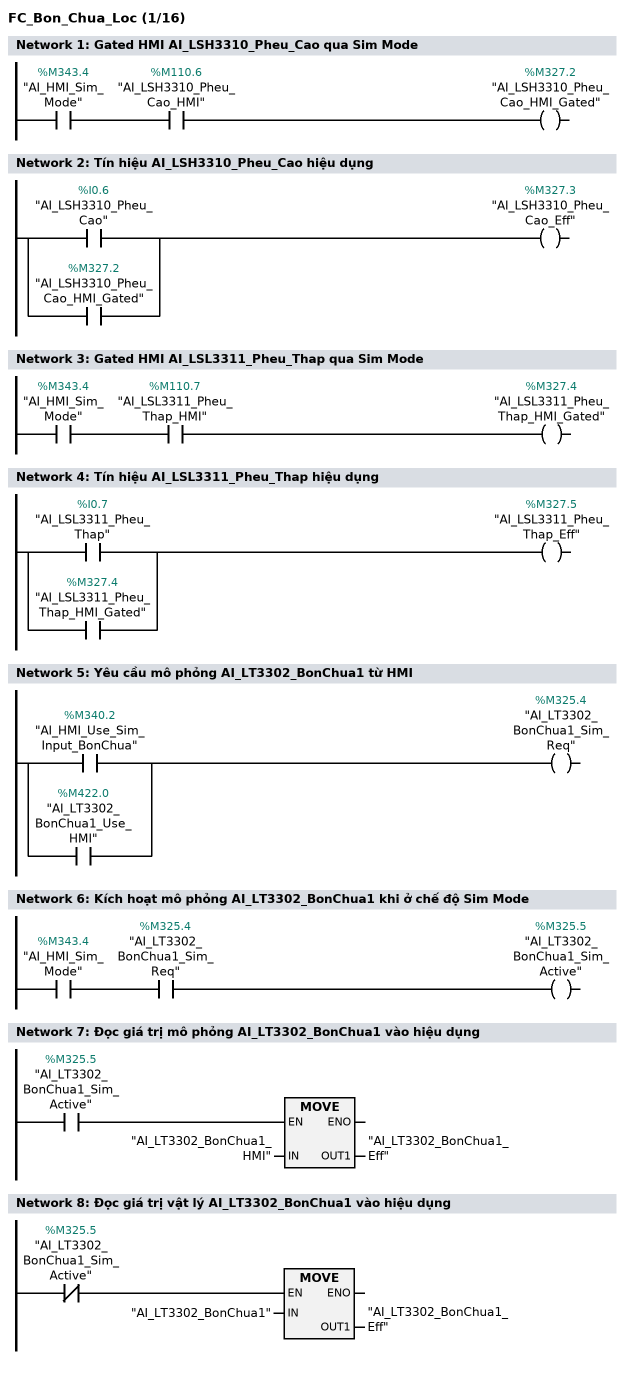
   RUNG wire#powerrail
      Contact( "AI_HMI_Sim_Mode" )
      Contact( "AI_LSH3310_Pheu_Cao_HMI" )
      Coil( "AI_LSH3310_Pheu_Cao_HMI_Gated" )
   END_RUNG
   // the same network as SCL:
   "AI_LSH3310_Pheu_Cao_HMI_Gated" := "AI_HMI_Sim_Mode" AND "AI_LSH3310_Pheu_Cao_HMI";
END_REGION

REGION Network 2: Tín hiệu AI_LSH3310_Pheu_Cao hiệu dụng
   RUNG wire#powerrail
      Contact( "AI_LSH3310_Pheu_Cao" )
      wire#w1
      Coil( "AI_LSH3310_Pheu_Cao_Eff" )
   END_RUNG
   RUNG wire#powerrail
      Contact( "AI_LSH3310_Pheu_Cao_HMI_Gated" )
   END_RUNG wire#w1
   // the same network as SCL:
   "AI_LSH3310_Pheu_Cao_Eff" := "AI_LSH3310_Pheu_Cao" OR "AI_LSH3310_Pheu_Cao_HMI_Gated";
END_REGION

REGION Network 3: Gated HMI AI_LSL3311_Pheu_Thap qua Sim Mode
   RUNG wire#powerrail
      Contact( "AI_HMI_Sim_Mode" )
      Contact( "AI_LSL3311_Pheu_Thap_HMI" )
      Coil( "AI_LSL3311_Pheu_Thap_HMI_Gated" )
   END_RUNG
   // the same network as SCL:
   "AI_LSL3311_Pheu_Thap_HMI_Gated" := "AI_HMI_Sim_Mode" AND "AI_LSL3311_Pheu_Thap_HMI";
END_REGION

REGION Network 4: Tín hiệu AI_LSL3311_Pheu_Thap hiệu dụng
   RUNG wire#powerrail
      Contact( "AI_LSL3311_Pheu_Thap" )
      wire#w1
      Coil( "AI_LSL3311_Pheu_Thap_Eff" )
   END_RUNG
   RUNG wire#powerrail
      Contact( "AI_LSL3311_Pheu_Thap_HMI_Gated" )
   END_RUNG wire#w1
   // the same network as SCL:
   "AI_LSL3311_Pheu_Thap_Eff" := "AI_LSL3311_Pheu_Thap" OR "AI_LSL3311_Pheu_Thap_HMI_Gated";
END_REGION

REGION Network 5: Yêu cầu mô phỏng AI_LT3302_BonChua1 từ HMI
   RUNG wire#powerrail
      Contact( "AI_HMI_Use_Sim_Input_BonChua" )
      wire#w1
      Coil( "AI_LT3302_BonChua1_Sim_Req" )
   END_RUNG
   RUNG wire#powerrail
      Contact( "AI_LT3302_BonChua1_Use_HMI" )
   END_RUNG wire#w1
   // the same network as SCL:
   "AI_LT3302_BonChua1_Sim_Req" := "AI_HMI_Use_Sim_Input_BonChua" OR "AI_LT3302_BonChua1_Use_HMI";
END_REGION

REGION Network 6: Kích hoạt mô phỏng AI_LT3302_BonChua1 khi ở chế độ Sim Mode
   RUNG wire#powerrail
      Contact( "AI_HMI_Sim_Mode" )
      Contact( "AI_LT3302_BonChua1_Sim_Req" )
      Coil( "AI_LT3302_BonChua1_Sim_Active" )
   END_RUNG
   // the same network as SCL:
   "AI_LT3302_BonChua1_Sim_Active" := "AI_HMI_Sim_Mode" AND "AI_LT3302_BonChua1_Sim_Req";
END_REGION

REGION Network 7: Đọc giá trị mô phỏng AI_LT3302_BonChua1 vào hiệu dụng
   RUNG wire#powerrail
      Contact( "AI_LT3302_BonChua1_Sim_Active" )
      { S7_GenerateENO := "TRUE" } Move(in := "AI_LT3302_BonChua1_HMI", out1 => "AI_LT3302_BonChua1_Eff")
   END_RUNG
   // the same network as SCL:
   IF "AI_LT3302_BonChua1_Sim_Active" THEN "AI_LT3302_BonChua1_Eff" := "AI_LT3302_BonChua1_HMI"; END_IF;
END_REGION

REGION Network 8: Đọc giá trị vật lý AI_LT3302_BonChua1 vào hiệu dụng
   RUNG wire#powerrail
      I_Contact( "AI_LT3302_BonChua1_Sim_Active" )
      { S7_GenerateENO := "TRUE" } Move(in := "AI_LT3302_BonChua1", out1 => "AI_LT3302_BonChua1_Eff")
   END_RUNG
   // the same network as SCL:
   IF NOT "AI_LT3302_BonChua1_Sim_Active" THEN "AI_LT3302_BonChua1_Eff" := "AI_LT3302_BonChua1"; END_IF;
END_REGION

REGION Network 9: Yêu cầu mô phỏng AI_TT3301_BonChua1 từ HMI
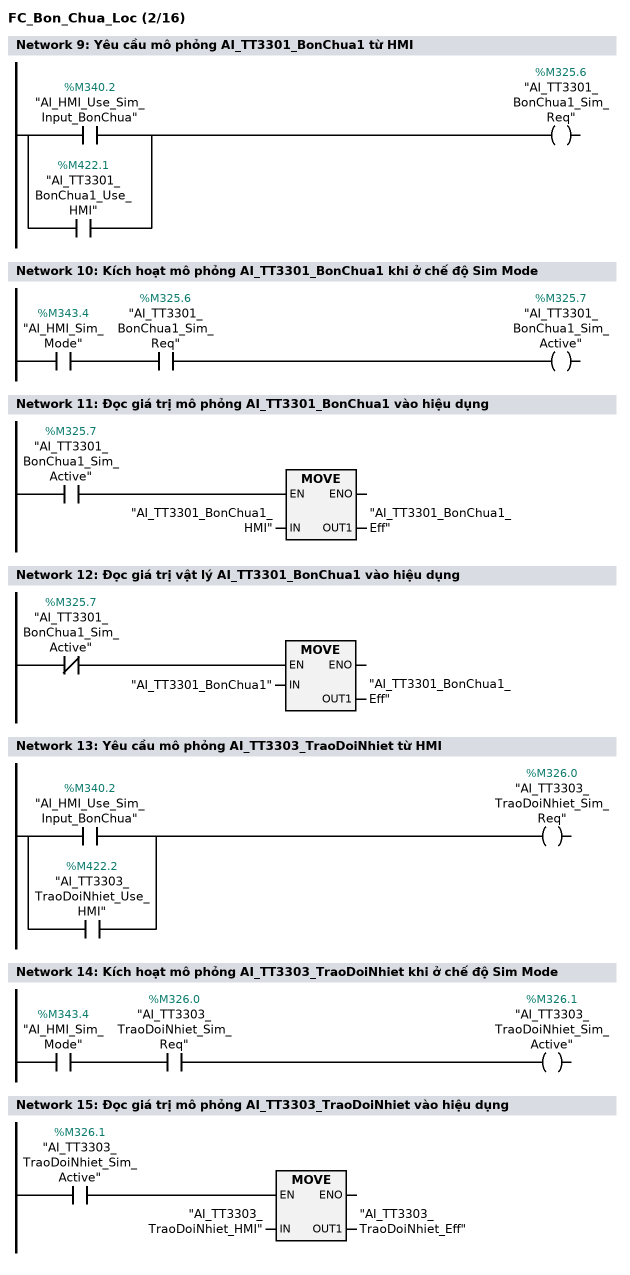
   RUNG wire#powerrail
      Contact( "AI_HMI_Use_Sim_Input_BonChua" )
      wire#w1
      Coil( "AI_TT3301_BonChua1_Sim_Req" )
   END_RUNG
   RUNG wire#powerrail
      Contact( "AI_TT3301_BonChua1_Use_HMI" )
   END_RUNG wire#w1
   // the same network as SCL:
   "AI_TT3301_BonChua1_Sim_Req" := "AI_HMI_Use_Sim_Input_BonChua" OR "AI_TT3301_BonChua1_Use_HMI";
END_REGION

REGION Network 10: Kích hoạt mô phỏng AI_TT3301_BonChua1 khi ở chế độ Sim Mode
   RUNG wire#powerrail
      Contact( "AI_HMI_Sim_Mode" )
      Contact( "AI_TT3301_BonChua1_Sim_Req" )
      Coil( "AI_TT3301_BonChua1_Sim_Active" )
   END_RUNG
   // the same network as SCL:
   "AI_TT3301_BonChua1_Sim_Active" := "AI_HMI_Sim_Mode" AND "AI_TT3301_BonChua1_Sim_Req";
END_REGION

REGION Network 11: Đọc giá trị mô phỏng AI_TT3301_BonChua1 vào hiệu dụng
   RUNG wire#powerrail
      Contact( "AI_TT3301_BonChua1_Sim_Active" )
      { S7_GenerateENO := "TRUE" } Move(in := "AI_TT3301_BonChua1_HMI", out1 => "AI_TT3301_BonChua1_Eff")
   END_RUNG
   // the same network as SCL:
   IF "AI_TT3301_BonChua1_Sim_Active" THEN "AI_TT3301_BonChua1_Eff" := "AI_TT3301_BonChua1_HMI"; END_IF;
END_REGION

REGION Network 12: Đọc giá trị vật lý AI_TT3301_BonChua1 vào hiệu dụng
   RUNG wire#powerrail
      I_Contact( "AI_TT3301_BonChua1_Sim_Active" )
      { S7_GenerateENO := "TRUE" } Move(in := "AI_TT3301_BonChua1", out1 => "AI_TT3301_BonChua1_Eff")
   END_RUNG
   // the same network as SCL:
   IF NOT "AI_TT3301_BonChua1_Sim_Active" THEN "AI_TT3301_BonChua1_Eff" := "AI_TT3301_BonChua1"; END_IF;
END_REGION

REGION Network 13: Yêu cầu mô phỏng AI_TT3303_TraoDoiNhiet từ HMI
   RUNG wire#powerrail
      Contact( "AI_HMI_Use_Sim_Input_BonChua" )
      wire#w1
      Coil( "AI_TT3303_TraoDoiNhiet_Sim_Req" )
   END_RUNG
   RUNG wire#powerrail
      Contact( "AI_TT3303_TraoDoiNhiet_Use_HMI" )
   END_RUNG wire#w1
   // the same network as SCL:
   "AI_TT3303_TraoDoiNhiet_Sim_Req" := "AI_HMI_Use_Sim_Input_BonChua" OR "AI_TT3303_TraoDoiNhiet_Use_HMI";
END_REGION

REGION Network 14: Kích hoạt mô phỏng AI_TT3303_TraoDoiNhiet khi ở chế độ Sim Mode
   RUNG wire#powerrail
      Contact( "AI_HMI_Sim_Mode" )
      Contact( "AI_TT3303_TraoDoiNhiet_Sim_Req" )
      Coil( "AI_TT3303_TraoDoiNhiet_Sim_Active" )
   END_RUNG
   // the same network as SCL:
   "AI_TT3303_TraoDoiNhiet_Sim_Active" := "AI_HMI_Sim_Mode" AND "AI_TT3303_TraoDoiNhiet_Sim_Req";
END_REGION

REGION Network 15: Đọc giá trị mô phỏng AI_TT3303_TraoDoiNhiet vào hiệu dụng
   RUNG wire#powerrail
      Contact( "AI_TT3303_TraoDoiNhiet_Sim_Active" )
      { S7_GenerateENO := "TRUE" } Move(in := "AI_TT3303_TraoDoiNhiet_HMI", out1 => "AI_TT3303_TraoDoiNhiet_Eff")
   END_RUNG
   // the same network as SCL:
   IF "AI_TT3303_TraoDoiNhiet_Sim_Active" THEN
       "AI_TT3303_TraoDoiNhiet_Eff" := "AI_TT3303_TraoDoiNhiet_HMI";
   END_IF;
END_REGION

REGION Network 16: Đọc giá trị vật lý AI_TT3303_TraoDoiNhiet vào hiệu dụng
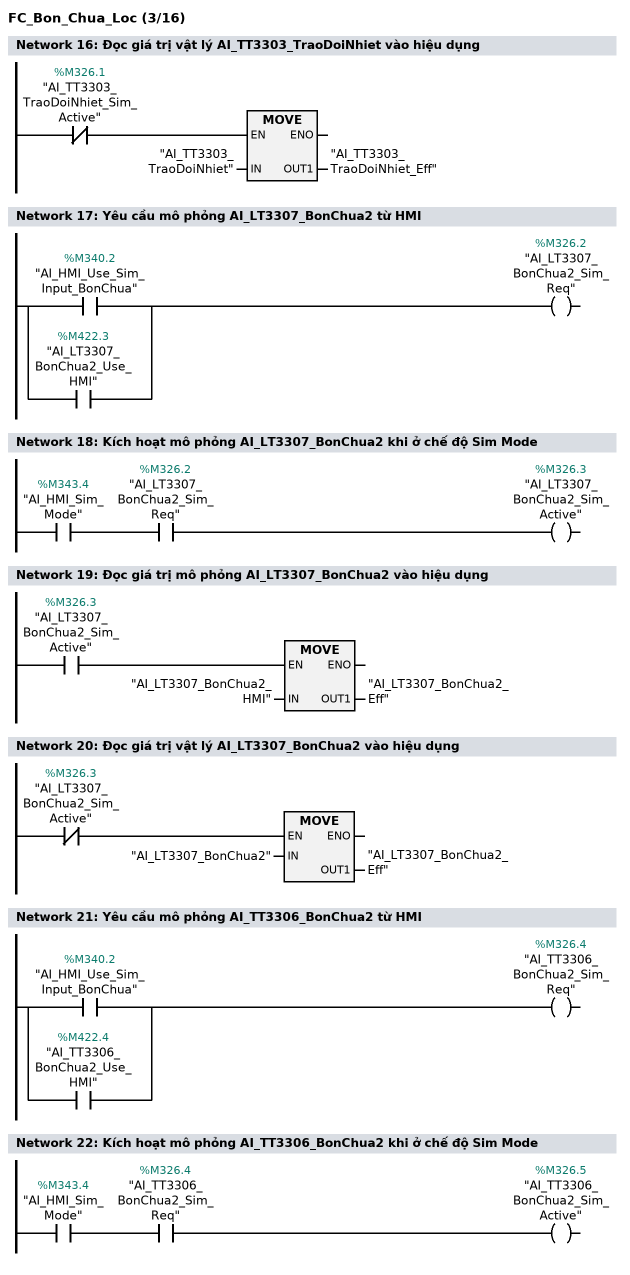
   RUNG wire#powerrail
      I_Contact( "AI_TT3303_TraoDoiNhiet_Sim_Active" )
      { S7_GenerateENO := "TRUE" } Move(in := "AI_TT3303_TraoDoiNhiet", out1 => "AI_TT3303_TraoDoiNhiet_Eff")
   END_RUNG
   // the same network as SCL:
   IF NOT "AI_TT3303_TraoDoiNhiet_Sim_Active" THEN
       "AI_TT3303_TraoDoiNhiet_Eff" := "AI_TT3303_TraoDoiNhiet";
   END_IF;
END_REGION

REGION Network 17: Yêu cầu mô phỏng AI_LT3307_BonChua2 từ HMI
   RUNG wire#powerrail
      Contact( "AI_HMI_Use_Sim_Input_BonChua" )
      wire#w1
      Coil( "AI_LT3307_BonChua2_Sim_Req" )
   END_RUNG
   RUNG wire#powerrail
      Contact( "AI_LT3307_BonChua2_Use_HMI" )
   END_RUNG wire#w1
   // the same network as SCL:
   "AI_LT3307_BonChua2_Sim_Req" := "AI_HMI_Use_Sim_Input_BonChua" OR "AI_LT3307_BonChua2_Use_HMI";
END_REGION

REGION Network 18: Kích hoạt mô phỏng AI_LT3307_BonChua2 khi ở chế độ Sim Mode
   RUNG wire#powerrail
      Contact( "AI_HMI_Sim_Mode" )
      Contact( "AI_LT3307_BonChua2_Sim_Req" )
      Coil( "AI_LT3307_BonChua2_Sim_Active" )
   END_RUNG
   // the same network as SCL:
   "AI_LT3307_BonChua2_Sim_Active" := "AI_HMI_Sim_Mode" AND "AI_LT3307_BonChua2_Sim_Req";
END_REGION

REGION Network 19: Đọc giá trị mô phỏng AI_LT3307_BonChua2 vào hiệu dụng
   RUNG wire#powerrail
      Contact( "AI_LT3307_BonChua2_Sim_Active" )
      { S7_GenerateENO := "TRUE" } Move(in := "AI_LT3307_BonChua2_HMI", out1 => "AI_LT3307_BonChua2_Eff")
   END_RUNG
   // the same network as SCL:
   IF "AI_LT3307_BonChua2_Sim_Active" THEN "AI_LT3307_BonChua2_Eff" := "AI_LT3307_BonChua2_HMI"; END_IF;
END_REGION

REGION Network 20: Đọc giá trị vật lý AI_LT3307_BonChua2 vào hiệu dụng
   RUNG wire#powerrail
      I_Contact( "AI_LT3307_BonChua2_Sim_Active" )
      { S7_GenerateENO := "TRUE" } Move(in := "AI_LT3307_BonChua2", out1 => "AI_LT3307_BonChua2_Eff")
   END_RUNG
   // the same network as SCL:
   IF NOT "AI_LT3307_BonChua2_Sim_Active" THEN "AI_LT3307_BonChua2_Eff" := "AI_LT3307_BonChua2"; END_IF;
END_REGION

REGION Network 21: Yêu cầu mô phỏng AI_TT3306_BonChua2 từ HMI
   RUNG wire#powerrail
      Contact( "AI_HMI_Use_Sim_Input_BonChua" )
      wire#w1
      Coil( "AI_TT3306_BonChua2_Sim_Req" )
   END_RUNG
   RUNG wire#powerrail
      Contact( "AI_TT3306_BonChua2_Use_HMI" )
   END_RUNG wire#w1
   // the same network as SCL:
   "AI_TT3306_BonChua2_Sim_Req" := "AI_HMI_Use_Sim_Input_BonChua" OR "AI_TT3306_BonChua2_Use_HMI";
END_REGION

REGION Network 22: Kích hoạt mô phỏng AI_TT3306_BonChua2 khi ở chế độ Sim Mode
   RUNG wire#powerrail
      Contact( "AI_HMI_Sim_Mode" )
      Contact( "AI_TT3306_BonChua2_Sim_Req" )
      Coil( "AI_TT3306_BonChua2_Sim_Active" )
   END_RUNG
   // the same network as SCL:
   "AI_TT3306_BonChua2_Sim_Active" := "AI_HMI_Sim_Mode" AND "AI_TT3306_BonChua2_Sim_Req";
END_REGION

REGION Network 23: Đọc giá trị mô phỏng AI_TT3306_BonChua2 vào hiệu dụng
